# B&R Automation Studio project HISTest (part 2)

#### mbus_mast.var - Local variables
```iecst
(********************************************************************
 * COPYRIGHT -- Bernecker + Rainer
 ********************************************************************
 * Program: mbus_mast
 * File: mbus_mast.var
 * Author: Bernecker + Rainer
 * Created: February 17, 2010
 ********************************************************************
 * Local variables of program mbus_mast
 ********************************************************************)
VAR
	step : step_typ;
END_VAR
```

#### Action.st
```iecst
ACTION ActMbRtuMaster:

	CASE step OF

		MB_OPEN:

			MbMaster.MBMOpen_0.enable	:= TRUE;

			//MbMaster.MBMOpen_0.pDevice	:= ADR('IF1.ST2.IF1.ST3.IF1');  (* Device description string *)

			MbMaster.MBMOpen_0.pDevice	:= ADR('IF6.ST1.IF1');
			MbMaster.MBMOpen_0.pMode	:= ADR('/PHY=RS485 /PA=N /DB=8 /SB=1 /BD=19200');  (* Mode description string *)
			MbMaster.MBMOpen_0.pConfig	:= ADR('datamod');  (* Data object name *)
			MbMaster.MBMOpen_0.timeout	:= 2000;  (* Timeout in milliseconds (the value must be a multiple of 10 and >250ms) *)
			MbMaster.MBMOpen_0.ascii	:= 0;  (* 0 = RTU / 1 = ASCII *)

			MbMaster.MBMOpen_0();

			IF (MbMaster.MBMOpen_0.status = 0) AND (MbMaster.MBMOpen_0.ident <> 0) THEN
				step := MB_RUN;
				gSignalCheck.RS485_Check := TRUE;
			ELSIF MbMaster.MBMOpen_0.status = 65535 THEN
			ELSIF MbMaster.MBMOpen_0.status <> 0 THEN
				step := MB_ERROR;
			END_IF

		MB_RUN:

			(*When the command Auto is True the MBMbMaster FUB is executed, otherwise the MCMCmd FUB is executed*)
			IF (MbMaster.Auto = TRUE) THEN
				MbMaster.MBMaster_0.enable	:= TRUE;
				MbMaster.MBMaster_0.ident		:= MbMaster.MBMOpen_0.ident;
				MbMaster.MBMaster_0();

				IF (MbMaster.MBMaster_0.status = 65535) THEN
				ELSIF MbMaster.MBMaster_0.status <> 0 THEN
					step := MB_ERROR;
				END_IF

			ELSE
				MbMaster.MBMCmd_0.enable	:= TRUE;
				MbMaster.MBMCmd_0.ident		:= MbMaster.MBMOpen_0.ident;

				IF (MbMaster.ReadDataTrigger) THEN
					MbMaster.MBMCmd_0.mfc 		:= 3;
					MbMaster.MBMCmd_0.data		:= ADR(MbMaster.ReadData);
					MbMaster.MBMCmd_0.offset	:= 0;
				ELSIF(MbMaster.WriteDataTrigger)THEN
					MbMaster.MBMCmd_0.mfc 		:= 16;
					MbMaster.MBMCmd_0.data		:= ADR(MbMaster.WriteData);  (* address of data area *)
					MbMaster.MBMCmd_0.offset	:= 100;
				END_IF;
				MbMaster.MBMCmd_0.node		:= 1;  (* address of the slave station *)
				MbMaster.MBMCmd_0.len		:= 10;
				MbMaster.MBMCmd_0();
				IF (MbMaster.MBMCmd_0.status = 65535) THEN
				ELSIF (MbMaster.MBMCmd_0.status <> 0) THEN
					step := MB_ERROR;
				END_IF

			END_IF

		MB_CLOSE:

			MbMaster.MBMClose_0.enable	:= TRUE;
			MbMaster.MBMClose_0.ident	:= MbMaster.MBMOpen_0.ident;
			MbMaster.MBMClose_0();

			IF MbMaster.MBMClose_0.status = 0 THEN
				step := MB_OPEN;
			ELSIF MbMaster.MBMClose_0.status = 65535 THEN
			ELSIF MbMaster.MBMClose_0.status <> 0 THEN
				step := MB_ERROR;
			END_IF

		MB_ERROR:

			MbMaster.MBMaster_0.enable	:= FALSE;
			MbMaster.MBMaster_0();
			MbMaster.MBMCmd_0.enable	:= FALSE;
			MbMaster.MBMCmd_0();
			MbMaster.MBMClose_0.enable	:= FALSE;
			MbMaster.MBMClose_0();

			IF (MbMaster.MBMOpen_0.ident <> 0) THEN
				MbMaster.MBMOpen_0.enable	:= FALSE;
				MbMaster.MBMOpen_0();
				step := MB_CLOSE;
			ELSE
				step := MB_OPEN;
			END_IF

	END_CASE

END_ACTION
```

### Data object Logical/MbRTU/datamod (Simple)

#### datamod.dat
```
(********************************************************************
 * COPYRIGHT -- Bernecker + Rainer
 ********************************************************************
 * Data object: NewDataObject
 * File: datamod.dat
 * Author: Bernecker + Rainer
 * Created: February 15, 2010
 ********************************************************************
 * Data object file: datamod.dat
 ********************************************************************)

;--------------------
; Modbus command file
;--------------------
"MbMaster.WriteDataTrigger      ", 16, $01, "MbMaster.WriteData             ", 00100, 0010
"MbMaster.ReadDataTrigger       ", 03, $01, "MbMaster.ReadData              ", 00000, 0010
"MbMaster.ReadDataTrigger       ", 03, $01, "MbMaster.ReadData              ", 00001, 0002

;"LibDRVmbus.EventPV4            ", 16, $01, "LibDRVmbus.LocalPV4            ", 0000, 0003
;"LibDRVmbus.EventPV3            ", 03, $01, "LibDRVmbus.LocalPV3            ", 0000, 0003
; \_____________________________/	|    |    \_____________________________/    |      |
;			 	 |					|    |				  	 |				     |      |
;		   31 Characters		    |    |			   31 Characters  		     |      |_Number of coils or registers
;			 						|    |				   						 |_Offset of the Modbus Variables
;									|    |
;									|    |_Target Address of the slave station
;			 						|
;			 						|_ Modbus function
```

### Program Logical/DIOHandle (IEC)

#### Variables.var
```iecst
VAR
	ProRLY : BOOL;
	PRLY : BOOL;
	NRLY : BOOL;
	ProRLYAUX : BOOL;
	PRLYAUX : BOOL;
	NRLYAUX : BOOL;
	EMSRLYAUX : BOOL;
END_VAR
```

#### Main.st
```iecst
PROGRAM _INIT
	(* Insert code here *)
	Sys.ProRly	:= 0;
	Sys.PRly	:= 0;
	Sys.NRly	:= 0;
	ProRLYAUX 	:= 0;
	PRLYAUX 	:= 0;
	NRLYAUX 	:= 0;
	EMSRLYAUX	:= 0;
END_PROGRAM

PROGRAM _CYCLIC
	(* Insert code here *)
	IF Sys.ProRly = 1	 	THEN
		ProRLY := 1;
	ELSE
	   	ProRLY := 0;
	END_IF;

	IF Sys.PRly = 1	 	THEN
		PRLY := 1;
	ELSE
		PRLY := 0;
	END_IF;

	IF Sys.NRly = 1	 	THEN
		NRLY := 1;
	ELSE
		NRLY := 0;
	END_IF;

	(* DI Check *)
	IF ProRLYAUX = 1 THEN
		Sys.ProRlyAux :=1;
	ELSE
		Sys.ProRlyAux :=0;
	END_IF;

	IF PRLYAUX = 1 THEN
		Sys.PRlyAux :=1;
	ELSE
		Sys.PRlyAux :=0;
	END_IF;

	IF NRLYAUX = 1 THEN
		Sys.NRlyAux :=1;
	ELSE
		Sys.NRlyAux :=0;
	END_IF;

	IF EMSRLYAUX = 1 THEN
		Sys.EMSRlyAux :=0;
	ELSE
		Sys.EMSRlyAux :=1;
	END_IF;

END_PROGRAM

PROGRAM _EXIT
	(* Insert code here *)

END_PROGRAM
```

### Program Logical/PRAHandle (IEC)

#### Variables.var
```iecst
VAR
	WakeUpSig : BOOL;
	PRATimerProRlyOff : TON;
	PRATimerProRlyOn : TON;
	PRATimerWakeUpOff : TON;
	PRATimerSeqErr : TON;
	LoopCount : USINT;
	RackIndex : USINT;
	WakeCount : USINT;
	RackCount : USINT;
END_VAR
```

#### Action.st
```iecst
ACTION ATSystemReady:

	PRARackEnableCount := 0;

	FOR i := 0 TO 3 DO
		IF SubBMS_Calculator.BSA[i].Rack_State.Field.BSA_Divice_Status <> 0 THEN
			PRARackEnableCount := PRARackEnableCount + 1 ;
		END_IF;
	END_FOR;

	IF PRARackEnableCount = HMI.DeviceLoading.SetRackNum THEN
		PRARackReadyDone := TRUE;
	ELSE
		PRARackReadyDone := FALSE;
	END_IF;
END_ACTION

ACTION ATReset:
	IF Sys.ResetSig THEN

		SubBMS_Calculator.BMA[0].Field.BSA_Reset := TRUE;
		SubBMS_Calculator.BMA[1].Field.BSA_Reset := TRUE;
		SubBMS_Calculator.BMA[2].Field.BSA_Reset := TRUE;
		SubBMS_Calculator.BMA[3].Field.BSA_Reset := TRUE;

		PRARackResetCount := 0;

		FOR i := 0 TO 3 DO
			IF SubBMS_Calculator.BSA[i].Rack_AlarmState.Value[1] = 0 AND SubBMS_Calculator.BSA[i].Rack_State.Field.BSA_Divice_Status <> 0 THEN
				PRARackResetCount := PRARackResetCount + 1 ;
			END_IF;
		END_FOR;

		IF PRARackResetCount = HMI.DeviceLoading.SetRackNum THEN
			PRARackResetDone := TRUE;
			PRATimerReset.IN := FALSE;

			SubBMS_Calculator.BMA[0].Field.BSA_Reset := FALSE;
			SubBMS_Calculator.BMA[1].Field.BSA_Reset := FALSE;
			SubBMS_Calculator.BMA[2].Field.BSA_Reset := FALSE;
			SubBMS_Calculator.BMA[3].Field.BSA_Reset := FALSE;

		ELSE
			PRARackResetDone := FALSE;
		END_IF;

	END_IF;

END_ACTION

ACTION ATWakeUpSeq:

	CASE WakeUpStep OF
		vkWAKEUP_INITIAL:

			Sys.WakeUpSig := TRUE;
			PRATimerSeqErr.IN := TRUE;

			IF 	Sys.WakeUpSig THEN
				WakeUpStep := vkWAKEUP_RACK1;
			END_IF;

		vkWAKEUP_RACK1: // RACK1 WakeUp

			SubBMS_Calculator.BMA[0].Field.BSA_WakeUP := TRUE;

			IF SubBMS_Calculator.BSA[0].Rack_State.Field.BSA_Divice_Status = 4 THEN
				WakeUpStep := vkWAKEUP_RACK2;
			ELSIF	SubBMS_Calculator.BSA[0].Rack_State.Field.BSA_Divice_Status = 0 THEN
				WakeUpStep := vkWAKEUP_RACK2;
				SubBMS_Calculator.BMA[0].Field.BSA_WakeUP := FALSE;
			END_IF;

		vkWAKEUP_RACK2: // RACK2 WakeUp

			SubBMS_Calculator.BMA[1].Field.BSA_WakeUP := TRUE;

			IF SubBMS_Calculator.BSA[1].Rack_State.Field.BSA_Divice_Status = 4 THEN
				WakeUpStep := vkWAKEUP_RACK3;
			ELSIF	SubBMS_Calculator.BSA[1].Rack_State.Field.BSA_Divice_Status = 0 THEN
				WakeUpStep := vkWAKEUP_RACK3;
				SubBMS_Calculator.BMA[1].Field.BSA_WakeUP := FALSE;
			END_IF;

		vkWAKEUP_RACK3: // RACK3 WakeUp

				SubBMS_Calculator.BMA[2].Field.BSA_WakeUP := TRUE;

			IF SubBMS_Calculator.BSA[2].Rack_State.Field.BSA_Divice_Status = 4  THEN
				WakeUpStep := vkWAKEUP_RACK4;
			ELSIF	SubBMS_Calculator.BSA[2].Rack_State.Field.BSA_Divice_Status = 0 THEN
				WakeUpStep := vkWAKEUP_RACK4;
				SubBMS_Calculator.BMA[2].Field.BSA_WakeUP := FALSE;
			END_IF;

		vkWAKEUP_RACK4: // RACK4 WakeUp

				SubBMS_Calculator.BMA[3].Field.BSA_WakeUP := TRUE;

			IF SubBMS_Calculator.BSA[3].Rack_State.Field.BSA_Divice_Status = 4 THEN
				WakeUpStep := vkWAKEUP_NRLY;
			ELSIF	SubBMS_Calculator.BSA[3].Rack_State.Field.BSA_Divice_Status = 0 THEN
				WakeUpStep := vkWAKEUP_NRLY;
				SubBMS_Calculator.BMA[3].Field.BSA_WakeUP := FALSE;
			END_IF;

		vkWAKEUP_NRLY: // SYSTEM NEG RLY ON

			Sys.NRly := 1;

			PMS.BAR_DIO.Field.BRA_Nrelay_DO_Status := TRUE;

			IF Sys.NRlyAux = 1 THEN
				WakeUpStep := vkWAKEUP_PRORLY_ON;
			END_IF;

		vkWAKEUP_PRORLY_ON: // SYSTEM PRO RLY ON

			Sys.ProRly :=1;

			PMS.BAR_DIO.Field.BRA_ProRelay_DO_Status := TRUE;

			IF Sys.ProRlyAux = 1 THEN
				WakeUpStep := vkWAKEUP_DELAYTIME1;
			END_IF;

		vkWAKEUP_DELAYTIME1: // DELAY TIME
			// Timmer1 on
			PRATimerProRlyOn.IN := TRUE;

			IF PRATimerProRlyOn.Q = 1 THEN
				WakeUpStep := vkWAKEUP_PRLY;
			END_IF;

		vkWAKEUP_PRLY: // SYSTEM POS RLY ON

			Sys.PRly :=1;

			PMS.BAR_DIO.Field.BRA_Prelay_DO_Status := TRUE;

			IF Sys.PRlyAux = 1 THEN
				WakeUpStep := vkWAKEUP_DELAYTIME2;
			END_IF;

		vkWAKEUP_DELAYTIME2 : // DELAY TIME
			// Timer2 on
			PRATimerProRlyOff.IN := TRUE;
			IF PRATimerProRlyOff.Q = 1 THEN
				WakeUpStep := vkWAKEUP_PRORLY_OFF;
			END_IF;

		vkWAKEUP_PRORLY_OFF: // SYSTEM PRO RLY OFF

			Sys.ProRly := 0;

			PMS.BAR_DIO.Field.BRA_ProRelay_DO_Status := FALSE;

			IF Sys.ProRlyAux = 0 THEN
				WakeUpStep := vkWAKEUP_TIMERESET;
			END_IF;

		vkWAKEUP_TIMERESET : // Timer reset

			PRATimerProRlyOn.IN 	:= FALSE;
			PRATimerProRlyOff.IN 	:= FALSE;
			PRATimerSeqErr.IN 		:= FALSE;

			Sys.WakeUpSig 	:= FALSE;
			PRAWakeUpDone 	:= TRUE;

	END_CASE;

END_ACTION
ACTION ATStopSeq:

	PRAStopDone 	:= FALSE;

	CASE StopStep OF
		vkSTOP_INITIAL:

			Sys.StopSig := TRUE;
			PRATimerSeqErr.IN := TRUE;

			IF Sys.StopSig THEN
				StopStep := vkSTOP_NRLY;
			END_IF;

		vkSTOP_NRLY: // SYSTEM NEG RLY ON

			Sys.NRly := 0;

			PMS.BAR_DIO.Field.BRA_Nrelay_DO_Status := FALSE;

			IF Sys.NRlyAux = 0 THEN
				StopStep := vkSTOP_DELAYTIME1;
			END_IF;

		vkSTOP_DELAYTIME1: // DELAY TIME
			// Timmer1 on
			PRATimerProRlyOn.IN := TRUE;
			IF PRATimerProRlyOn.Q = 1 THEN
				StopStep := vkSTOP_PRLY;
			END_IF;

		vkSTOP_PRLY: // SYSTEM POS RLY ON

			Sys.PRly := 0;

			PMS.BAR_DIO.Field.BRA_Prelay_DO_Status := FALSE;

			IF Sys.PRlyAux = 0 THEN
				StopStep := vkSTOP_DELAYTIME2;
			END_IF;

		vkSTOP_DELAYTIME2 : // DELAY TIME
			// Timer2 on
			PRATimerProRlyOff.IN := TRUE;
			IF PRATimerProRlyOff.Q = 1 THEN
				StopStep := vkSTOP_RACK1;
			END_IF;

		vkSTOP_RACK1: // RACK1 WakeUp

			IF SubBMS_Calculator.BSA[0].Rack_State.Field.BSA_Divice_Status = 4 THEN
				SubBMS_Calculator.BMA[0].Field.BSA_WakeUP := FALSE;
			END_IF;

			IF SubBMS_Calculator.BSA[0].Rack_State.Field.BSA_Divice_Status = 3 OR SubBMS_Calculator.BSA[0].Rack_State.Field.BSA_Divice_Status = 0 THEN
				StopStep := vkSTOP_RACK2;
			END_IF;

		vkSTOP_RACK2: // RACK2 WakeUp

			IF SubBMS_Calculator.BSA[1].Rack_State.Field.BSA_Divice_Status = 4 THEN
				SubBMS_Calculator.BMA[1].Field.BSA_WakeUP := FALSE;
			END_IF;

			IF SubBMS_Calculator.BSA[1].Rack_State.Field.BSA_Divice_Status = 3 OR SubBMS_Calculator.BSA[1].Rack_State.Field.BSA_Divice_Status = 0 THEN
				StopStep := vkSTOP_RACK3;
			END_IF;

		vkSTOP_RACK3: // RACK3 WakeUp

			IF SubBMS_Calculator.BSA[2].Rack_State.Field.BSA_Divice_Status = 4 THEN
				SubBMS_Calculator.BMA[2].Field.BSA_WakeUP := FALSE;
			END_IF;

			IF SubBMS_Calculator.BSA[2].Rack_State.Field.BSA_Divice_Status = 3 OR SubBMS_Calculator.BSA[2].Rack_State.Field.BSA_Divice_Status = 0 THEN
				StopStep := vkSTOP_RACK4;
			END_IF;

		vkSTOP_RACK4: // RACK4 WakeUp

			IF SubBMS_Calculator.BSA[3].Rack_State.Field.BSA_Divice_Status = 4 THEN
				SubBMS_Calculator.BMA[3].Field.BSA_WakeUP := FALSE;
			END_IF;

			IF SubBMS_Calculator.BSA[3].Rack_State.Field.BSA_Divice_Status = 3 OR SubBMS_Calculator.BSA[3].Rack_State.Field.BSA_Divice_Status = 0 THEN
				StopStep := vkSTOP_TIMERESET;
			END_IF;

		vkSTOP_TIMERESET : // Timer reset

			PRATimerWakeUpOff.IN	:= FALSE;
			PRATimerSeqErr.IN		:= FALSE;

			PRAStopDone 	:= TRUE;

	END_CASE;

END_ACTION
```

#### Main.st
```iecst
PROGRAM _INIT
	(* Insert code here *)
	StateMa := 0;

	RackIndex := 0;
	RackEnable_Count := 0;

	PRATimerProRlyOn.IN		:= FALSE;
	PRATimerProRlyOn.PT 	:= T#500ms;
	PRATimerProRlyOff.IN	:= FALSE;
	PRATimerProRlyOff.PT	:= T#200ms;
	PRATimerWakeUpOff.IN 	:= FALSE;
	PRATimerWakeUpOff.PT 	:= T#100ms;
	PRATimerSeqErr.IN 		:= FALSE;
	PRATimerSeqErr.PT 		:= T#15s;

END_PROGRAM

PROGRAM _CYCLIC
	(* Insert code here *)

//		 EMS EDGE POSITIVE TRIGGER 		//

//	IF EDGEPOS(Sys.EMSRlyAux) THEN
//	  StateMa := 14;
//	END_IF;
//
//

	CASE StateMa OF
		vkSYSTEM_INITIAL: // INITIAL

			IF HMI.DeviceLoading.SetRackNum <> 0 THEN
	  			StateMa		:= vkSYSTEM_PROTECT_CHECK;
			END_IF;

		vkSYSTEM_PROTECT_CHECK:

			IF HMI.DialogBox.Protect_Trigger THEN
				StateMa		:= vkSUBBMS_TEMPCHECK;
			ELSE
				StateMa		:= vkSUBBMS_ALLRESET;
			END_IF;

			RackIndex := 0;
			RackEnable_Count := 0;

		vkSUBBMS_ALLRESET: // SUB BMS ALL RESET COMMAND ON

			FOR LoopCount := 0  TO RACK_MAXNUM_MINUS_1 DO
				SubBMS_Calculator.BMA[LoopCount].Field.BSA_Reset := TRUE;
			END_FOR;

			StateMa := vkSUBBMS_STATECHECK;

		vkSUBBMS_STATECHECK: // SUB BMS STATE CHECK AND SUB BMS RESET COMMAND OFF

			IF (SubBMS_Calculator.BMA[RackIndex].Field.BSA_Reset) THEN

				IF SubBMS_Calculator.BSA[RackIndex].Rack_State.Field.BSA_Divice_Status <> 0 THEN
					SubBMS_Calculator.BMA[RackIndex].Field.BSA_Reset := FALSE;

					RackEnable_Count	:= RackEnable_Count + 1;

				ELSIF SubBMS_Calculator.BSA[RackIndex].Rack_State.Field.BSA_Divice_Status = 0 THEN

					SubBMS_Calculator.BMA[RackIndex].Field.BSA_Reset := FALSE;

				END_IF;

			END_IF;

			RackIndex := RackIndex + 1;

			IF RackIndex >= 4 THEN

				RackIndex	:= 0;

				IF RackEnable_Count = (HMI.DeviceLoading.SetRackNum) THEN
					StateMa := vkSUBBMS_WAITCOMMAND;
				END_IF;

			END_IF;

		vkSUBBMS_TEMPCHECK:

			IF SubBMS_Calculator.BSA[RackIndex].Rack_State.Field.BSA_Divice_Status <> 0 THEN

				RackEnable_Count	:= RackEnable_Count + 1;

			ELSIF SubBMS_Calculator.BSA[RackIndex].Rack_State.Field.BSA_Divice_Status = 0 THEN

			END_IF;

			RackIndex := RackIndex + 1;

			IF RackIndex >= 4 THEN

				RackIndex	:= 0;

				IF RackEnable_Count = (HMI.DeviceLoading.SetRackNum) THEN
					StateMa := vkSUBBMS_WAITCOMMAND;
				END_IF;

			END_IF;

		vkSUBBMS_WAITCOMMAND: // WAIT COMMAND
			IF (PMS.PMS.Field.PMS_WakeUp_CMD) AND NOT(PMS.PMS.Field.PMS_FaultReset) AND NOT(PMS.PMS.Field.PMS_Po_RelayStatus) AND NOT(PMS.PMS.Field.PMS_Pro_RelayStatus) AND NOT(PMS.PMS.Field.PMS_Ne_RelayStatus) AND ABS(PMS.SysBatCal.Field.BSA_Curr_Total) <= 50 THEN
				StateMa := vkSUBBMS_FIRSTWAKEUP;
			END_IF;

		vkSUBBMS_FIRSTWAKEUP: // INITIATE FIRST WAKE-UP
			PRATimerSeqErr.IN := TRUE;

			RackIndex := 0;
			WakeCount := 0;

			FOR LoopCount := 0  TO RACK_MAXNUM_MINUS_1 DO
				IF HMI.RackEnable[LoopCount] THEN
					SubBMS_Calculator.BMA[LoopCount].Field.BSA_WakeUP 	:= TRUE;
					RackIndex											:=	LoopCount;
					EXIT;
				END_IF;

			END_FOR;
			//SubBMS_Calculator.BMA[RackIndex].Field.BSA_WakeUP := TRUE;

			StateMa := vkSUBBMS_WAKEUPSEQ;

		vkSUBBMS_WAKEUPSEQ: // CHECK CURRENT RACK STATUS

			IF SubBMS_Calculator.BSA[RackIndex].Rack_State.Field.BSA_Divice_Status = 4 THEN

				WakeCount := WakeCount + 1;

				IF RackIndex <= RACK_MAXNUM_MINUS_1-1 THEN
					FOR LoopCount := RackIndex + 1  TO RACK_MAXNUM_MINUS_1 DO
						IF HMI.RackEnable[LoopCount] THEN
							SubBMS_Calculator.BMA[LoopCount].Field.BSA_WakeUP 	:= TRUE;
							RackIndex											:=	LoopCount;
							EXIT;
						END_IF;

					END_FOR;
				END_IF;

				IF WakeCount = RackEnable_Count THEN
					StateMa := vkSYSTEM_NEGRLY_ON;
				ELSE
					IF WakeCount > RACK_MAXNUM_MINUS_1 THEN
						WakeCount	:= 0;
					END_IF;
				END_IF;
			END_IF;

		vkSYSTEM_NEGRLY_ON: // SYSTEM NEG RLY ON
			Sys.NRly := 1;

			PMS.BAR_DIO.Field.BRA_Nrelay_DO_Status := TRUE;

			IF Sys.NRlyAux = 1 THEN
	  			StateMa := vkSYSTEM_PRORLY_ON;
			END_IF;

		vkSYSTEM_PRORLY_ON: // SYSTEM PRO RLY ON
			Sys.ProRly :=1;

			PMS.BAR_DIO.Field.BRA_ProRelay_DO_Status := TRUE;

			IF Sys.ProRlyAux = 1 THEN
	  			StateMa := vkSYSTEM_RLYDELAY1;
			END_IF;

		vkSYSTEM_RLYDELAY1: // DELAY TIME
			// Timmer1 on
			PRATimerProRlyOn.IN := TRUE;
			IF PRATimerProRlyOn.Q = 1 THEN
				StateMa := vkSYSTEM_POSRLY_ON;
			END_IF;

		vkSYSTEM_POSRLY_ON: // SYSTEM POS RLY ON
			Sys.PRly :=1;

			PMS.BAR_DIO.Field.BRA_Prelay_DO_Status := TRUE;

			IF Sys.PRlyAux = 1 THEN
	  			StateMa := vkSYSTEM_RLYDELAY2;
			END_IF;

		vkSYSTEM_RLYDELAY2 : // DELAY TIME
			// Timer2 on
			PRATimerProRlyOff.IN := TRUE;
			IF PRATimerProRlyOff.Q = 1 THEN
				StateMa := vkSYSTEM_PRORLY_OFF;
			END_IF;

		vkSYSTEM_PRORLY_OFF: // SYSTEM PRO RLY OFF
			Sys.ProRly := 0;

			PMS.BAR_DIO.Field.BRA_ProRelay_DO_Status := FALSE;

			IF Sys.ProRlyAux = 0 THEN
	  			StateMa := vkSYSTEM_DELAY_RESET1;
			END_IF;

		vkSYSTEM_DELAY_RESET1 : // Timer reset

			PRATimerProRlyOn.IN 	:= FALSE;
			PRATimerProRlyOff.IN 	:= FALSE;
			PRATimerSeqErr.IN 		:= FALSE;

			StateMa := vkSYSTEM_RUN;

		vkSYSTEM_RUN: //RUN STATE (IDLE)

			IF NOT(PMS.PMS.Field.PMS_WakeUp_CMD) AND NOT(PMS.PMS.Field.PMS_FaultReset) AND NOT(PMS.PMS.Field.PMS_Po_RelayStatus) AND NOT(PMS.PMS.Field.PMS_Pro_RelayStatus) AND NOT(PMS.PMS.Field.PMS_Ne_RelayStatus) AND ABS(PMS.SysBatCal.Field.BSA_Curr_Total) <= 50 THEN
				StateMa := vkSYSTEM_NEGRLY_OFF;
			END_IF;
		vkSYSTEM_NEGRLY_OFF:

			PRATimerSeqErr.IN := TRUE;

			Sys.NRly := 0;

			PMS.BAR_DIO.Field.BRA_Nrelay_DO_Status := FALSE;

			IF Sys.NRlyAux = 0 THEN
				StateMa := vkSYSTEM_RLYDELAY3;
			END_IF;

		vkSYSTEM_RLYDELAY3 :
			PRATimerWakeUpOff.IN := TRUE;
			IF PRATimerWakeUpOff.Q = 1 THEN
				StateMa := vkSYSTEM_POSRLY_OFF;
			END_IF;

		vkSYSTEM_POSRLY_OFF :
			Sys.PRly := 0;

			PMS.BAR_DIO.Field.BRA_Prelay_DO_Status := FALSE;

			IF Sys.PRlyAux = 0 THEN
				StateMa := vkSUBBMS_FIRSTWAKEDOWN;
			END_IF;

		vkSUBBMS_FIRSTWAKEDOWN: // INITIATE FIRST WAKE-UP

			RackIndex := 0;
			WakeCount := 0;

			FOR LoopCount := 0  TO RACK_MAXNUM_MINUS_1 DO
				IF HMI.RackEnable[LoopCount] THEN
					SubBMS_Calculator.BMA[LoopCount].Field.BSA_WakeUP 	:= FALSE;
					RackIndex											:=	LoopCount;
					EXIT;
				END_IF;

			END_FOR;
			//SubBMS_Calculator.BMA[RackIndex].Field.BSA_WakeUP := TRUE;
			StateMa := vkSUBBMS_WAKEDOWNSEQ;

		vkSUBBMS_WAKEDOWNSEQ: // CHECK CURRENT RACK STATUS

			IF SubBMS_Calculator.BSA[RackIndex].Rack_State.Field.BSA_Divice_Status = 3 THEN

				WakeCount := WakeCount + 1;

				IF RackIndex <= RACK_MAXNUM_MINUS_1-1 THEN
					FOR LoopCount := RackIndex + 1  TO RACK_MAXNUM_MINUS_1 DO
						IF HMI.RackEnable[LoopCount] THEN
							SubBMS_Calculator.BMA[LoopCount].Field.BSA_WakeUP 	:= FALSE;
							RackIndex											:=	LoopCount;
							EXIT;
						END_IF;

					END_FOR;
				END_IF;

				IF WakeCount = RackEnable_Count THEN
					StateMa := vkSYSTEM_DELAY_RESET2;
				ELSE
					IF WakeCount > RACK_MAXNUM_MINUS_1 THEN
	 					WakeCount	:= 0;
					END_IF;

				END_IF;
			END_IF;
//			IF SubBMS_Calculator.BSA[RackIndex].Rack_State.Field.BSA_Divice_Status = 3 THEN
//				RackIndex := RackIndex + 1;
//
//				IF RackIndex <= Rack_Count THEN
//					SubBMS_Calculator.BMA[RackIndex].Field.BSA_WakeUP := FALSE;
//
//					StateMa := 18;
//				ELSE
//
//					StateMa := 19;
//				END_IF;
//			END_IF;

		vkSYSTEM_DELAY_RESET2 :
			PRATimerWakeUpOff.IN	:= FALSE;
			PRATimerSeqErr.IN		:= FALSE;

			StateMa := vkSUBBMS_WAITCOMMAND;

	END_CASE;

	// SYSTEM STATE SEQ AND RELAY CHECK

	CASE StateMa OF
		0..4: // RESET SEQ

			IF RackCount = HMI.DeviceLoading.SetRackNum THEN

				PMS.SysBatCal.Field.BSA_Divice_Status := 1; //INIT

			ELSE

				FOR LoopCount := 0  TO RACK_MAXNUM_MINUS_1 DO
					IF (HMI.RackEnable[LoopCount]) THEN
						IF SubBMS_Calculator.BSA[LoopCount].Rack_State.Field.BSA_Divice_Status = 3 OR  SubBMS_Calculator.BSA[LoopCount].Rack_State.Field.BSA_Divice_Status = 2 THEN
							RackCount := RackCount + 1 ;
						END_IF;
					END_IF;
				END_FOR;

				PMS.SysBatCal.Field.BSA_Divice_Status := 0; //READY

			END_IF;

			IF PMS.PMS.Field.PMS_Po_RelayStatus OR PMS.PMS.Field.PMS_Pro_RelayStatus OR PMS.PMS.Field.PMS_Ne_RelayStatus THEN
				PMS.BAR_Protect.Field.BRA_Prtct_RelayWelding := TRUE;
			ELSE
				PMS.BAR_Protect.Field.BRA_Prtct_RelayWelding := FALSE;
			END_IF;

		5:
			FOR LoopCount := 0 TO RACK_MAXNUM_MINUS_1 DO
				IF SubBMS_Calculator.BSA[LoopCount].Rack_State.Field.BSA_Neg_Rly OR SubBMS_Calculator.BSA[LoopCount].Rack_State.Field.BSA_Pos_Rly OR SubBMS_Calculator.BSA[LoopCount].Rack_State.Field.BSA_PreChar_Rly THEN
	  				PMS.BAR_Protect.Field.BRA_Prtct_RelayWelding := TRUE;
				END_IF;

			END_FOR;

			IF Sys.PRly OR Sys.NRly OR Sys.ProRly THEN
				PMS.BAR_Protect.Field.BRA_Prtct_RelayWelding := TRUE;
			ELSE
				PMS.BAR_Protect.Field.BRA_Prtct_RelayWelding := FALSE;
			END_IF;

		6..14: //WAKE UP SEQ
			PMS.SysBatCal.Field.BSA_Divice_Status := 2; //STANDBY

			IF PRATimerSeqErr.Q = 1 THEN
				//PMS.PMS_PAR_SEQErr := TRUE;
			END_IF;

		15:
			IF PMS.PMS.Field.PMS_Po_RelayStatus AND NOT(PMS.PMS.Field.PMS_Pro_RelayStatus) AND PMS.PMS.Field.PMS_Ne_RelayStatus THEN
				PMS.SysBatCal.Field.BSA_Divice_Status := 3; //RUN
			END_IF;

		16..21: //WAKE DOWN SEQ

			IF NOT(Sys.NRly) AND NOT(Sys.PRly) THEN
				PMS.SysBatCal.Field.BSA_Divice_Status := 2; //STANDBY
			END_IF;

			IF PRATimerSeqErr.Q = 1 THEN
				//PMS.PMS_PAR_SEQErr := TRUE;
			END_IF;

	END_CASE;

	PRATimerProRlyOn();
	PRATimerProRlyOff();
	PRATimerWakeUpOff();
	PRATimerSeqErr();

END_PROGRAM

PROGRAM _EXIT
	(* Insert code here *)

END_PROGRAM
```

### SubBMS.typ
```iecst
TYPE
	SubBMS_Calculator_type : 	STRUCT
		BMA : ARRAY[0..3]OF BMAN_typ;
		BSA : ARRAY[0..3]OF BSA_typ;
	END_STRUCT;
	SubBMS_type : 	STRUCT
		Rack1 : SubBMS_Rack_type;
		Rack2 : SubBMS_Rack_type;
		Rack3 : SubBMS_Rack_type;
		Rack4 : SubBMS_Rack_type;
	END_STRUCT;
	SubBMS_Rack_type : 	STRUCT
		BMA : BMAN_typ;
		BSA : BSA_typ;
	END_STRUCT;
	BMA_typ : 	STRUCT
		BMA1 : BMAN_typ;
		BMA2 : BMAN_typ;
		BMA3 : BMAN_typ;
		BMA4 : BMAN_typ;
	END_STRUCT;
	BMAN_typ : 	STRUCT
		Value : ARRAY[0..1]OF DWORD;
		Field : BMAN_Field_typ;
	END_STRUCT;
	BMAN_Field_typ : 	STRUCT
		BSA_WakeUP : BOOL;
		BSA_Mode : BOOL;
		BSA_Reset : BOOL;
		BSA_Cell_MinV : UINT;
		BSA_Cell_AGV : INT;
	END_STRUCT;
	BSA_typ : 	STRUCT
		BSA_Product : BSA_Product_typ;
		Rack_Calc : Rack_Calc_typ;
		Rack_State : Rack_State_typ;
		Rack_AlarmState : Rack_AlarmState_typ;
		Rack_PWRCalc : Rack_PWRCalc_typ;
		Rack_Cell_Vcalc : Rack_Cell_Vcalc_typ;
		Rack_Cell_Tcalc : Rack_Cell_Tcalc_typ;
		Rack_Cell_Pcalc : Rack_Cell_Pcalc_typ;
		Modul1_Info : ModulN_Info_typ;
		Modul2_Info : ModulN_Info_typ;
		Modul3_Info : ModulN_Info_typ;
		Modul4_Info : ModulN_Info_typ;
		Modul5_Info : ModulN_Info_typ;
		Modul6_Info : ModulN_Info_typ;
		Modul7_Info : ModulN_Info_typ;
	END_STRUCT;
	BSA_Product_typ : 	STRUCT
		Value : ARRAY[0..1]OF DWORD;
		Field : BSA_Product_Field_typ;
	END_STRUCT;
	Rack_Calc_typ : 	STRUCT
		Value : ARRAY[0..1]OF DWORD;
		Field : Rack_Calc_Field_typ;
	END_STRUCT;
	Rack_State_typ : 	STRUCT
		Value : ARRAY[0..1]OF DWORD;
		Field : Rack_State_Field_typ;
	END_STRUCT;
	Rack_AlarmState_typ : 	STRUCT
		Value : ARRAY[0..1]OF DWORD;
		Field : Rack_AlarmState_Fieild_typ;
	END_STRUCT;
	Rack_PWRCalc_typ : 	STRUCT
		Value : ARRAY[0..1]OF DWORD;
		Field : Rack_PWRCalc_Field_typ;
	END_STRUCT;
	Rack_Cell_Vcalc_typ : 	STRUCT
		Value : ARRAY[0..1]OF DWORD;
		Field : Rack_Cell_Vcalc_Field_typ;
	END_STRUCT;
	Rack_Cell_Tcalc_typ : 	STRUCT
		Value : ARRAY[0..1]OF DWORD;
		Field : Rack_Cell_Tcalc_Field_typ;
	END_STRUCT;
	Rack_Cell_Pcalc_typ : 	STRUCT
		Value : ARRAY[0..1]OF DWORD;
		Field : Rack_Cell_Pcalc_Field_typ;
	END_STRUCT;
	ModulN_Info_typ : 	STRUCT
		Value : ARRAY[0..1]OF DWORD;
		Field : ModulN_Info_Field_typ;
	END_STRUCT;
	BSA_Product_Field_typ : 	STRUCT
		BSA_Type : USINT;
		BSA_SW_Ver : USINT;
		BRA_Normal_Volt : REAL;
		BRA_Capacity : REAL;
		BSA_Serial : USINT;
		BSA_Parallel : USINT;
	END_STRUCT;
	Rack_Calc_Field_typ : 	STRUCT
		BRA_Volt_Total : REAL;
		BRA_Curr_Total : REAL;
		BRA_SOC : REAL;
		BRA_SOH : REAL;
	END_STRUCT;
	Rack_State_Field_typ : 	STRUCT
		BSA_Divice_Status : USINT;
		BSA_Protect_Status : USINT;
		BSA_Balance : BOOL;
		BSA_Neg_Rly : BOOL;
		BSA_Pos_Rly : BOOL;
		BSA_PreChar_Rly : BOOL;
		BSA_MSD_AUX : BOOL;
		BSA_EMG_SW : BOOL;
		BSA_Water_leak : BOOL;
		Not_Used1 : BOOL;
		Not_Used2 : USINT;
		BSA_Ah : INT;
		Not_Used3 : UINT;
	END_STRUCT;
	Rack_AlarmState_Fieild_typ : 	STRUCT
		warning : Rack_warningState_Field_typ;
		fault : Rack_FaultState_Field_typ;
		protect : Rack_ProtectState_Field_typ;
	END_STRUCT;
	Rack_warningState_Field_typ : 	STRUCT
		BSA_Wn_Dischager_OC : BOOL;
		BSA_Wn_Chager_OC : BOOL;
		BSA_Wn_SOC_OV : BOOL;
		BSA_Wn_SOC_Un : BOOL;
		BSA_Wn_OV : BOOL;
		BSA_Wn_UV : BOOL;
		BSA_Wn_Cell_OV : BOOL;
		BSA_Wn_Cell_UV : BOOL;
		BSA_Wn_Cell_UnbalV : BOOL;
		BSA_Wn_DisCharger_Cell_OT : BOOL;
		BSA_Wn_Charger_Cell_OT : BOOL;
		BSA_Wn_DisCharger_Cell_UT : BOOL;
		BSA_Wn_Charger_Cell_UT : BOOL;
		BSA_Wn_Cell_UnbalT : BOOL;
		BSA_Wn_Discharger_UnbaPWR : BOOL;
		BSA_Wn_Charger_UnbaPWR : BOOL;
	END_STRUCT;
	Rack_FaultState_Field_typ : 	STRUCT
		BSA_FLT_Dischager_OC : BOOL;
		BSA_FLT_Chager_OC : BOOL;
		BSA_FLT_SOC_OV : BOOL;
		BSA_FLT_SOC_Un : BOOL;
		BSA_FLT_OV : BOOL;
		BSA_FLT_UV : BOOL;
		BSA_FLT_Cell_OV : BOOL;
		BSA_FLT_Cell_UV : BOOL;
		BSA_FLT_Cell_UnbalV : BOOL;
		BSA_FLT_DisCharger_Cell_OT : BOOL;
		BSA_FLT_Charger_Cell_OT : BOOL;
		BSA_FLT_DisCharger_Cell_UT : BOOL;
		BSA_FLT_Charger_Cell_UT : BOOL;
		BSA_FLT_Cell_UnbalT : BOOL;
		BSA_FLT_Discharger_UnbaPWR : BOOL;
		BSA_FLT_Charger_UnbaPWR : BOOL;
	END_STRUCT;
	Rack_ProtectState_Field_typ : 	STRUCT
		BSA_Prtct_Dischager_OC : BOOL;
		BSA_Prtct_Chager_OC : BOOL;
		BSA_Prtct_SOC_OV : BOOL;
		BSA_Prtct_SOC_Un : BOOL;
		BSA_Prtct_OV : BOOL;
		BSA_Prtct_UV : BOOL;
		BSA_Prtct_Cell_OV : BOOL;
		BSA_Prtct_Cell_UV : BOOL;
		BSA_Prtct_Cell_UnbalV : BOOL;
		BSA_Prtct_DisCharger_Cell_OT : BOOL;
		BSA_Prtct_Charger_Cell_OT : BOOL;
		BSA_Prtct_DisCharger_Cell_UT : BOOL;
		BSA_Prtct_Charger_Cell_UT : BOOL;
		BSA_Prtct_Cell_UnbalT : BOOL;
		BSA_Prtct_Discharger_UnbaPWR : BOOL;
		BSA_Prtct_Charger_UnbaPWR : BOOL;
		BSA_Prtct_Rly_Err : BOOL;
		BSA_Prtct_IN_COM_Err : BOOL;
		BSA_Prtct_EX_COM_Err : BOOL;
		BSA_Prtct_CT_COM_Err : BOOL;
		BSA_Prtct_Water_Leak_Err : BOOL;
		BSA_Prtct_EMS_SW_Err : BOOL;
		Not_Used1 : BOOL;
		Not_Used2 : BOOL;
		Not_Used3 : USINT;
	END_STRUCT;
	Rack_PWRCalc_Field_typ : 	STRUCT
		BSA_CHAPWCont : REAL;
		BSA_DisCHAPWCont : REAL;
		BSA_CHAPWPeak : REAL;
		BSA_DisCHAPWPeak : REAL;
	END_STRUCT;
	Rack_Cell_Vcalc_Field_typ : 	STRUCT
		BSA_Cell_MaxV : REAL;
		BSA_Cell_MinV : REAL;
		BSA_Cell_AVGV : REAL;
		BSA_Cell_DeviV : UINT;
	END_STRUCT;
	Rack_Cell_Tcalc_Field_typ : 	STRUCT
		BSA_Cell_MaxT : REAL;
		BSA_Cell_MinT : REAL;
		BSA_Cell_AVGT : REAL;
		BSA_Cell_DeviT : REAL;
	END_STRUCT;
	Rack_Cell_Pcalc_Field_typ : 	STRUCT
		BSA_Cell_MaxV_Location : UINT;
		BSA_Cell_MinV_Location : UINT;
		BSA_Cell_MaxT_Location : UINT;
		BSA_Cell_MinT_Location : UINT;
	END_STRUCT;
	ModulN_Info_Field_typ : 	STRUCT
		Volt_Total : REAL;
		Agv_Volt : REAL;
		Agv_Temp : REAL;
		OPS_INITOK : BOOL;
		OPS_Fault : BOOL;
		OPS_Balan_On_OFF : BOOL;
		OPS_Waterleak_Err : BOOL;
		OPS_CellVolt_Err : BOOL;
		OPS_CellTemps_Err : BOOL;
		BATIC_Err : BOOL;
		CTCOM_Err : BOOL;
		OPS_MBCOM_Err : BOOL;
		Not_Used1 : BOOL;
		Not_Used2 : BOOL;
		Not_Used3 : BOOL;
		Not_Used4 : BOOL;
		Not_Used5 : BOOL;
		Not_Used6 : BOOL;
		Not_Used7 : BOOL;
	END_STRUCT;
END_TYPE
```

### HMI.typ
```iecst
TYPE
	HMI_typ : 	STRUCT
		Step : STEP_Enum;
		DeviceLoading : DeviceLoadingPanel_typ;
		RackEnable : ARRAY[0..RACK_MAXNUM_MINUS_1]OF BOOL;
		RackIndex : RackIndex_enum;
		Gauge : GaugePanel_typ;
		BatteryInfo : BATInfoPanel_typ;
		Module1Info : ModuleInfoPanel_typ;
		Module2Info : ModuleInfoPanel_typ;
		Module3Info : ModuleInfoPanel_typ;
		Module4Info : ModuleInfoPanel_typ;
		Module5Info : ModuleInfoPanel_typ;
		Module6Info : ModuleInfoPanel_typ;
		Module7Info : ModuleInfoPanel_typ;
		SystemRackInfo : SystemRackInfoPanel_typ;
		BSA_Divice_Status : STRING[20];
		DIOStatus : DIOStatusPanel_typ;
		ProtectStatus : ProtectStatusPanel_typ;
		SubBMS_AlarmTable : ARRAY[0..21]OF ALARM_Info_typ;
		AlarmTableIndex : AlarmTableIndex_enum;
		AdminLogin : AdminLogin_typ;
		AdminDeviceReset : BOOL;
		TrendData : TrendData_typ;
		DialogBox : DialogBox_typ;
	END_STRUCT;
	DeviceLoadingPanel_typ : 	STRUCT
		Trigger : BOOL;
		DeviceLoadingStep : USINT;
		RackLoading : USINT;
		DeviceLoading_Max : USINT;
		SetRackNum : USINT;
		LoadingText : STRING[40];
	END_STRUCT;
	GaugePanel_typ : 	STRUCT
		BRA_SOC : REAL;
		BRA_SOC_A : STRING[20];
		BRA_SOC_B : STRING[50];
		BRA_SOH : REAL;
		BRA_SOH_A : STRING[20];
		BRA_SOH_B : STRING[50];
		BRA_Volt_Total : REAL;
		BRA_Volt_Total_A : STRING[20];
		BRA_Volt_Total_B : STRING[50];
		BRA_Curr_Total : REAL;
		BRA_Curr_Total_A : STRING[20];
		BRA_Curr_Total_B : STRING[50];
	END_STRUCT;
	BATInfoPanel_typ : 	STRUCT
		BSA_Cell_MaxV : REAL;
		BSA_Cell_MinV : REAL;
		BSA_Cell_AVGV : REAL;
		BSA_Cell_DeviV : REAL;
		BSA_Cell_MaxT : REAL;
		BSA_Cell_MinT : REAL;
		BSA_Cell_AVGT : REAL;
		BSA_Cell_DeviT : REAL;
		BSA_Cell_MaxV_Rack_Location : STRING[20];
		BSA_Cell_MaxV_Cell_Location : STRING[20];
		BSA_Cell_MaxV_Location : STRING[20];
		BSA_Cell_MinV_Rack_Location : STRING[20];
		BSA_Cell_MinV_Cell_Location : STRING[20];
		BSA_Cell_MinV_Location : STRING[20];
		BSA_Cell_MaxT_Rack_Location : STRING[20];
		BSA_Cell_MaxT_Cell_Location : STRING[20];
		BSA_Cell_MaxT_Location : STRING[20];
		BSA_Cell_MinT_Rack_Location : STRING[20];
		BSA_Cell_MinT_Cell_Location : STRING[20];
		BSA_Cell_MinT_Location : STRING[20];
	END_STRUCT;
	ModuleInfoPanel_typ : 	STRUCT
		Volt_Total_A : STRING[20];
		Volt_Total_B : STRING[20];
		OPS_Fault : STRING[20];
		CTCOM_Err : STRING[20];
		OPS_MBCOM_Err : STRING[20];
	END_STRUCT;
	SystemRackInfoPanel_typ : 	STRUCT
		RACK_State : ARRAY[0..3]OF STRING[20];
		RACK_BRA_Volt_Total : ARRAY[0..3]OF STRING[20];
		RACK_BRA_Curr_Total : ARRAY[0..3]OF STRING[20];
		RACK_BRA_Total : ARRAY[0..3]OF STRING[20];
	END_STRUCT;
	DIOStatusPanel_typ : 	STRUCT
		BSA_EMS : STRING[20];
		BSA_OffGas : STRING[20];
		BSA_Water_leak : STRING[20];
		BSA_Neg_Rly : STRING[20];
		BSA_PreChar_Rly : STRING[20];
		BSA_Pos_Rly : STRING[20];
	END_STRUCT;
	ProtectStatusPanel_typ : 	STRUCT
		BSA_Charge_OC : STRING[20];
		BSA_Discharge_OC : STRING[20];
		BSA_OC : STRING[20];
		BSA_SOC_OV : STRING[20];
		BSA_SOC_Un : STRING[20];
		BSA_OV : STRING[20];
		BSA_UV : STRING[20];
		BSA_Cell_OV : STRING[20];
		BSA_Cell_UV : STRING[20];
		BSA_Cell_UnbalV : STRING[20];
		BSA_DisCharger_Cell_OT : STRING[20];
		BSA_Charger_Cell_OT : STRING[20];
		BSA_DisCharger_Cell_UT : STRING[20];
		BSA_Charger_Cell_UT : STRING[20];
		BSA_Cell_UnbalT : STRING[20];
		BSA_Discharge_Unbal_PWR : STRING[20];
		BSA_Charge_Unbal_PWR : STRING[20];
		BSA_Prtct_Peak_OP : STRING[20];
		BSA_Prtct_Continuously_OP : STRING[20];
		BSA_Prtct_IN_COM_Err : STRING[20];
		BSA_Prtct_EX_COM_Err : STRING[20];
		BSA_Prtct_Rly_Err : STRING[20];
		BSA_Prtct_Water_Leak_Err : STRING[20];
		BRA_Prtct_InsulationReg : STRING[20];
		BRA_Prtct_MDSFuse : STRING[20];
		BSA_Prtct_CoolingSystem : STRING[20];
	END_STRUCT;
	Alarm_typ : 	STRUCT
		Warning : ARRAY[0..21]OF ALARM_Info_typ;
		Fault : ARRAY[0..21]OF ALARM_Info_typ;
		Protect : ARRAY[0..21]OF ALARM_Info_typ;
	END_STRUCT;
	ALARM_Info_typ : 	STRUCT
		Name : STRING[30];
		InitialTime : STRING[15];
		RecentTime : STRING[15];
		ClearTime : STRING[15];
		Count : USINT;
	END_STRUCT;
	Dialog_typ : 	STRUCT
		Name : STRING[30];
		Trigger : BOOL;
	END_STRUCT;
	AdminLogin_typ : 	STRUCT
		Authority : LoginStatusEnum;
		Input_Button : STRING[1];
		Password_Internal : STRING[16];
		Password_External : STRING[16];
	END_STRUCT;
	TrendData_typ : 	STRUCT
		Voltage : REAL;
		Current : REAL;
	END_STRUCT;
	DialogBox_typ : 	STRUCT
		LoadingError_Trigger : BOOL;
		BuzzerOFF_Trigger : BOOL;
		Protect_Trigger : BOOL;
		ProtectName : STRING[30];
	END_STRUCT;
	STEP_Enum :
		(
		vkINITIAL := 0,
		vkBOOTING := 1,
		vkSYSTEM := 2,
		vkRACK1 := 3,
		vkRACK2 := 4,
		vkRACK3 := 5,
		vkRACK4 := 6,
		vkADMINISTRATOR := 13,
		vkALARMHISTORY := 14,
		vkLOADINGERROR := 15,
		vkPROTECTERROR := 16,
		vkUSERTEST := 20
		);
	RackIndex_enum :
		(
		vkRACKNUM1 := 0,
		vkRACKNUM2 := 1,
		vkRACKNUM3 := 2,
		vkRACKNUM4 := 3
		);
	AlarmTableIndex_enum :
		(
		vkWarning := 0,
		vkFault := 1,
		vkProtect := 2
		);
	LoginStatusEnum :
		(
		USER := 0,
		ADMIN := 1
		);
END_TYPE
```

### PMS_CAN.typ
```iecst
TYPE
	PMS_typ : 	STRUCT
		PMS : PMS_type;
		SysBatProduct : SysBatProduct_typ;
		SysBatCal : SysBatCal_typ;
		SysBatPWR : SysBatPWR_typ;
		SysCellVolt : SysCellVolt_typ;
		SysCellTemps : SysCellTemps_typ;
		SysCellV_TPos : SysCellV_TPos_typ;
		SysBatProtect : SysBatProtect_typ;
		SysBatDIO : SysBatDIO_typ;
		BRACal : BRACal_typ;
		BRAPWR_A : BRAPWR_A_typ;
		BRAPWR_B : BRAPWR_B_typ;
		BRACellV : BRACellV_typ;
		BRACellT : BRACellT_typ;
		BRACellDiv : BRACellDiv_typ;
		BRA_VTPos : BRA_VTPos_typ;
		BAR_Alarm : BAR_Alarm_typ;
		BAR_Protect : BAR_Protect_typ;
		BAR_DIO : BAR_DIO_typ;
	END_STRUCT;
	PMS_type : 	STRUCT
		Value : ARRAY[0..1]OF DWORD;
		Field : PMS_Field_typ;
	END_STRUCT;
	SysBatProduct_typ : 	STRUCT
		Value : ARRAY[0..1]OF DWORD;
		Field : SysBatProduct_Field_typ;
	END_STRUCT;
	SysBatCal_typ : 	STRUCT
		Value : ARRAY[0..1]OF DWORD;
		Field : SysBatCal_Field_typ;
	END_STRUCT;
	SysBatPWR_typ : 	STRUCT
		Value : ARRAY[0..1]OF DWORD;
		Field : SysBatPWR_Field_typ;
	END_STRUCT;
	SysCellVolt_typ : 	STRUCT
		Value : ARRAY[0..1]OF DWORD;
		Field : SysCellVolt_Field_typ;
	END_STRUCT;
	SysCellTemps_typ : 	STRUCT
		Value : ARRAY[0..1]OF DWORD;
		Field : SysCellTemps_Field_typ;
	END_STRUCT;
	SysCellV_TPos_typ : 	STRUCT
		Value : ARRAY[0..1]OF DWORD;
		Field : SysCellV_TPos_Field_typ;
	END_STRUCT;
	SysBatProtect_typ : 	STRUCT
		Value : ARRAY[0..1]OF DWORD;
		Field : SysBatProtect_Field_typ;
	END_STRUCT;
	SysBatDIO_typ : 	STRUCT
		Value : ARRAY[0..1]OF DWORD;
		Field : SysBatDIO_Field_typ;
	END_STRUCT;
	BRACal_typ : 	STRUCT
		Value : ARRAY[0..1]OF DWORD;
		Field : BRACal_Field_typ;
	END_STRUCT;
	BRAPWR_A_typ : 	STRUCT
		Value : ARRAY[0..1]OF DWORD;
		Field : BRAPWR_A_Field_typ;
	END_STRUCT;
	BRAPWR_B_typ : 	STRUCT
		Value : ARRAY[0..1]OF DWORD;
		Field : BRAPWR_B_Field_typ;
	END_STRUCT;
	BRACellV_typ : 	STRUCT
		Value : ARRAY[0..1]OF DWORD;
		Field : BRACellV_Field_typ;
	END_STRUCT;
	BRACellT_typ : 	STRUCT
		Value : ARRAY[0..1]OF DWORD;
		Field : BRACellT_Field_typ;
	END_STRUCT;
	BRACellDiv_typ : 	STRUCT
		Value : ARRAY[0..1]OF DWORD;
		Field : BRACellDiv_Field_typ;
	END_STRUCT;
	BRA_VTPos_typ : 	STRUCT
		Value : ARRAY[0..1]OF DWORD;
		Field : BRA_VTPos_Field_typ;
	END_STRUCT;
	BAR_Alarm_typ : 	STRUCT
		Value : ARRAY[0..1]OF DWORD;
		Field : BAR_Alarm_Field_typ;
	END_STRUCT;
	BAR_Protect_typ : 	STRUCT
		Value : ARRAY[0..1]OF DWORD;
		Field : BAR_Protect_Field_typ;
	END_STRUCT;
	BAR_DIO_typ : 	STRUCT
		Value : ARRAY[0..1]OF DWORD;
		Field : BAR_DIO_Field_typ;
	END_STRUCT;
	PMS_Field_typ : 	STRUCT
		PMS_WakeUp_CMD : BOOL;
		PMS_POWER_CMD : BOOL;
		PMS_FaultReset : BOOL;
		PMS_Po_RelayStatus : BOOL;
		PMS_Pro_RelayStatus : BOOL;
		PMS_Ne_RelayStatus : BOOL;
	END_STRUCT;
	SysBatProduct_Field_typ : 	STRUCT
		BSA_Production_Year : UINT;
		BSA_Production_Type : USINT;
		BSA_Production_Num : USINT;
		BSA_Production_VER : USINT;
		BSA_Production_BSA_Serial : USINT;
		BSA_Production_BSA_Parallel : USINT;
	END_STRUCT;
	SysBatCal_Field_typ : 	STRUCT
		BSA_Volt_Total : REAL;
		BSA_Curr_Total : REAL;
		BSA_SOC : REAL;
		BSA_Divice_Status : UINT;
	END_STRUCT;
	SysBatPWR_Field_typ : 	STRUCT
		BSA_Cont_Charge_Power_Limit : REAL;
		BSA_Peak_Charge_Power_Limit : REAL;
		BSA_Cont_Discharge_Power_Limit : REAL;
		BSA_Peak_Discharge_Power_Limit : REAL;
	END_STRUCT;
	SysCellVolt_Field_typ : 	STRUCT
		BSA_Cell_MaxV : REAL;
		BSA_Cell_MinV : REAL;
		BSA_Cell_AVGV : REAL;
		BSA_Cell_DeviV : REAL;
	END_STRUCT;
	SysCellTemps_Field_typ : 	STRUCT
		BSA_Cell_MaxT : REAL;
		BSA_Cell_MinT : REAL;
		BSA_Cell_AVGT : REAL;
		BSA_Cell_DeviT : REAL;
	END_STRUCT;
	SysCellV_TPos_Field_typ : 	STRUCT
		BSA_Rack_MaxV_Location : USINT;
		BSA_Cell_MaxV_Location : USINT;
		BSA_Rack_MinV_Location : USINT;
		BSA_Cell_MinV_Location : USINT;
		BSA_Rack_MaxT_Location : USINT;
		BSA_Cell_MaxT_Location : USINT;
		BSA_Rack_MinT_Location : USINT;
		BSA_Cell_MinT_Location : USINT;
	END_STRUCT;
	SysBatProtect_Field_typ : 	STRUCT
		BSA_Alarm_OC : BOOL;
		BSA_Alarm_SOC_OV : BOOL;
		BSA_Alarm_SOC_UN : BOOL;
		BSA_Alarm_OV : BOOL;
		BSA_Alarm_UV : BOOL;
		BSA_Alarm_Cell_OV : BOOL;
		BSA_Alarm_Cell_UV : BOOL;
		BSA_Alarm_Cell_UnBalaV : BOOL;
		BSA_Alarm_Discharger_Cell_OT : BOOL;
		BSA_Alarm_Charger_Cell_OT : BOOL;
		BSA_Alarm_Discharger_Cell_UT : BOOL;
		BSA_Alarm_Charger_Cell_UT : BOOL;
		BSA_Alarm_Cell_UnBalaT : BOOL;
		BSA_Alarm_Continuously_OP : BOOL;
		BSA_Alarm_Peak_OP : BOOL;
		BSA_Fault_OC : BOOL;
		BSA_Fault_SOC_OV : BOOL;
		BSA_Fault_SOC_UN : BOOL;
		BSA_Fault_OV : BOOL;
		BSA_Fault_UV : BOOL;
		BSA_Fault_Cell_OV : BOOL;
		BSA_Fault_Cell_UV : BOOL;
		BSA_Fault_Cell_UnBalaV : BOOL;
		BSA_Fault_Discharger_Cell_OT : BOOL;
		BSA_Fault_Charger_Cell_OT : BOOL;
		BSA_Fault_Discharger_Cell_UT : BOOL;
		BSA_Fault_Charger_Cell_UT : BOOL;
		BSA_Fault_Cell_UnBalaT : BOOL;
		BSA_Fault_Continuously_OP : BOOL;
		BSA_Fault_Peak_OP : BOOL;
		BSA_Prtct_OC : BOOL;
		BSA_Prtct_SOC_OV : BOOL;
		BSA_Prtct_SOC_UN : BOOL;
		BSA_Prtct_OV : BOOL;
		BSA_Prtct_UV : BOOL;
		BSA_Prtct_Cell_OV : BOOL;
		BSA_Prtct_Cell_UV : BOOL;
		BSA_Prtct_Cell_UnBalaV : BOOL;
		BSA_Prtct_Discharger_Cell_OT : BOOL;
		BSA_Prtct_Charger_Cell_OT : BOOL;
		BSA_Prtct_Discharger_Cell_UT : BOOL;
		BSA_Prtct_Charger_Cell_UT : BOOL;
		BSA_Prtct_Cell_UnBalaT : BOOL;
		BSA_Prtct_Continuously_OP : BOOL;
		BSA_Prtct_Peak_OP : BOOL;
		BSA_Prtct_InternalCOM : BOOL;
		BSA_Prtct_ExternalCOM : BOOL;
		BSA_Prtct_RelayWelding : BOOL;
		BSA_Prtct_WaterLeak : BOOL;
		BSA_Prtct_InsulationReg : BOOL;
		BSA_Prtct_MDSFuse : BOOL;
		BSA_Prtct_Cooling_System : BOOL;
	END_STRUCT;
	SysBatDIO_Field_typ : 	STRUCT
		BSA_Prelay_DO_Status : BOOL;
		BSA_Nrelay_DO_Status : BOOL;
		BSA_ProRelay_DO_Status : BOOL;
		BSA_Buzzer_DO_Status : BOOL;
		BSA_PowerLamp_DO_Status : BOOL;
		BSA_DO_Spare06 : BOOL;
		BSA_DO_Spare07 : BOOL;
		BSA_DO_Spare08 : BOOL;
		BSA_DO_Spare09 : BOOL;
		BSA_DO_Spare10 : BOOL;
		BSA_DO_Spare11 : BOOL;
		BSA_DO_Spare12 : BOOL;
		BSA_PRelayAUX_DI_Status : BOOL;
		BSA_NRelayAUX_DI_Status : BOOL;
		BSA_EMGSwitch_DI_Status : BOOL;
		BSA_CoolingSystem_DI_Status : BOOL;
		BSA_MDS_DI_Status : BOOL;
		BSA_DI_Spare06 : BOOL;
		BSA_DI_Spare07 : BOOL;
		BSA_DI_Spare08 : BOOL;
		BSA_DI_Spare09 : BOOL;
		BSA_DI_Spare10 : BOOL;
		BSA_DI_Spare11 : BOOL;
		BSA_DI_Spare12 : BOOL;
		BSA_SOH : REAL;
	END_STRUCT;
	BRACal_Field_typ : 	STRUCT
		BRA_Rack_Num : UINT;
		BRA_Volt_Total : REAL;
		BRA_Curr_Total : REAL;
		BRA_SOC : REAL;
	END_STRUCT;
	BRAPWR_A_Field_typ : 	STRUCT
		BRA_Rack_Num : UINT;
		BRA_SOH : REAL;
		BRA_CONT_CHA_PWR_Limit : REAL;
		BRA_Peak_CHA_PWR_Limit : REAL;
	END_STRUCT;
	BRAPWR_B_Field_typ : 	STRUCT
		BRA_Rack_Num : UINT;
		BRA_CONT_DisCHA_PWR_Limit : REAL;
		BRA_Peak_DisCHA_PWR_Limit : REAL;
	END_STRUCT;
	BRACellV_Field_typ : 	STRUCT
		BRA_Rack_Num : UINT;
		BRA_Cell_Max_Voltage : REAL;
		BRA_Cell_Min_Voltage : REAL;
		BRA_Cell_AGV_Voltage : REAL;
	END_STRUCT;
	BRACellT_Field_typ : 	STRUCT
		BRA_Rack_Num : UINT;
		BRA_Cell_Max_Temperature : REAL;
		BRA_Cell_Min_Temperature : REAL;
		BRA_Cell_AGV_Temperature : REAL;
	END_STRUCT;
	BRACellDiv_Field_typ : 	STRUCT
		BRA_Rack_Num : UINT;
		BRA_Cell_DIV_Voltage : REAL;
		BRA_Cell_DIV_Temperature : REAL;
	END_STRUCT;
	BRA_VTPos_Field_typ : 	STRUCT
		BRA_Rack_Num : UINT;
		BRA_Max_Cell_V_Location : USINT;
		BRA_Min_Cell_V_Location : USINT;
		BRA_Max_Cell_T_Location : USINT;
		BRA_Min_Cell_T_Location : USINT;
	END_STRUCT;
	BAR_Alarm_Field_typ : 	STRUCT
		BRA_Rack_Num : UINT;
		BRA_Alarm_OC : BOOL;
		BRA_Alarm_SOC_OV : BOOL;
		BRA_Alarm_SOC_UN : BOOL;
		BRA_Alarm_OV : BOOL;
		BRA_Alarm_UV : BOOL;
		BRA_Alarm_Cell_OV : BOOL;
		BRA_Alarm_Cell_UV : BOOL;
		BRA_Alarm_Cell_UnBalaV : BOOL;
		BRA_Alarm_Discharger_Cell_OT : BOOL;
		BRA_Alarm_Charger_Cell_OT : BOOL;
		BRA_Alarm_Discharger_Cell_UT : BOOL;
		BRA_Alarm_Charger_Cell_UT : BOOL;
		BRA_Alarm_Cell_UnBalaT : BOOL;
		BRA_Alarm_Continuously_OP : BOOL;
		BRA_Alarm_Peak_OP : BOOL;
		BRA_Fault_OC : BOOL;
		BRA_Fault_SOC_OV : BOOL;
		BRA_Fault_SOC_UN : BOOL;
		BRA_Fault_OV : BOOL;
		BRA_Fault_UV : BOOL;
		BRA_Fault_Cell_OV : BOOL;
		BRA_Fault_Cell_UV : BOOL;
		BRA_Fault_Cell_UnBalaV : BOOL;
		BRA_Fault_Discharger_Cell_OT : BOOL;
		BRA_Fault_Charger_Cell_OT : BOOL;
		BRA_Fault_Discharger_Cell_UT : BOOL;
		BRA_Fault_Charger_Cell_UT : BOOL;
		BRA_Fault_Cell_UnBalaT : BOOL;
		BRA_Fault_Continuously_OP : BOOL;
		BRA_Fault_Peak_OP : BOOL;
	END_STRUCT;
	BAR_Protect_Field_typ : 	STRUCT
		BRA_Rack_Num : UINT;
		BRA_Prtct_OC : BOOL;
		BRA_Prtct_SOC_OV : BOOL;
		BRA_Prtct_SOC_UN : BOOL;
		BRA_Prtct_OV : BOOL;
		BRA_Prtct_UV : BOOL;
		BRA_Prtct_Cell_OV : BOOL;
		BRA_Prtct_Cell_UV : BOOL;
		BRA_Prtct_Cell_UnBalaV : BOOL;
		BRA_Prtct_Discharger_Cell_OT : BOOL;
		BRA_Prtct_Charger_Cell_OT : BOOL;
		BRA_Prtct_Discharger_Cell_UT : BOOL;
		BRA_Prtct_Charger_Cell_UT : BOOL;
		BRA_Prtct_Cell_UnBalaT : BOOL;
		BRA_Prtct_Continuously_OP : BOOL;
		BRA_Prtct_Peak_OP : BOOL;
		BRA_Prtct_InternalCOM : BOOL;
		BRA_Prtct_ExternalCOM : BOOL;
		BRA_Prtct_RelayWelding : BOOL;
		BRA_Prtct_WaterLeak : BOOL;
		BRA_Prtct_InsulationReg : BOOL;
		BRA_Prtct_MDSFuse : BOOL;
		BRA_Prtct_CoolingSystem : BOOL;
	END_STRUCT;
	BAR_DIO_Field_typ : 	STRUCT
		BRA_Rack_Num : UINT;
		BRA_Prelay_DO_Status : BOOL;
		BRA_Nrelay_DO_Status : BOOL;
		BRA_ProRelay_DO_Status : BOOL;
		BRA_PowerLamp_DO_Status : BOOL;
		BRA_Buzzer_DO_Status : BOOL;
		BRA_PRelayAUX_DI_Status : BOOL;
		BRA_NRelayAUX_DI_Status : BOOL;
		BRA_EMGSwitch_DI_Status : BOOL;
		BRA_MDS_DI_Status : BOOL;
		BRA_Waterleak_Dete_MD1 : BOOL;
		BRA_Waterleak_Dete_MD2 : BOOL;
		BRA_Waterleak_Dete_MD3 : BOOL;
		BRA_Waterleak_Dete_MD4 : BOOL;
		BRA_Waterleak_Dete_MD5 : BOOL;
		BRA_Waterleak_Dete_MD6 : BOOL;
		BRA_Waterleak_Dete_MD7 : BOOL;
	END_STRUCT;
END_TYPE
```

### LAMP.typ
```iecst
TYPE
	LAMP_typ : 	STRUCT
		SW_B : BOOL;
	END_STRUCT;
END_TYPE
```

### Variables.var
```iecst
VAR CONSTANT
	PASSWORD : STRING[16] := '1234';
	RACK1 : USINT := 0;
	RACK2 : USINT := 1;
	RACK3 : USINT := 2;
	RACK4 : USINT := 3;
	RACK_MAXNUM : USINT := 4;
	RACK_MAXNUM_MINUS_1 : USINT := RACK_MAXNUM-1;
END_VAR
(*Insert your comment here.*)
(*Insert your comment here.*)
(*Insert your comment here.*)
VAR
	SubBMS : SubBMS_type;
	SubBMS_Sim : SubBMS_type;
	SubBMS_Calculator : SubBMS_Calculator_type;
	Rack_HMI : BSA_typ;
END_VAR
(*Insert your comment here.*)
(*Insert your comment here.*)
(*Insert your comment here.*)
VAR
	HMI : HMI_typ;
END_VAR
VAR RETAIN
	HMI_Alarm : Alarm_typ;
	HMI_AlarmName : ARRAY[0..21] OF STRING[30];
END_VAR
VAR
	HMI_Dialog : Dialog_typ;
END_VAR
(*Insert your comment here.*)
(*Insert your comment here.*)
(*Insert your comment here.*)
VAR
	PMS : PMS_typ;
	System_HMI : PMS_typ;
END_VAR
(*Insert your comment here.*)
(*Insert your comment here.*)
(*Insert your comment here.*)
VAR
	LAMP : LAMP_typ;
END_VAR
```

### Program Logical/Source/LAMPSeq/Lamp_SW_B (IEC)

#### Main.st
```iecst
PROGRAM _INIT
	(* Insert code here *)

END_PROGRAM

PROGRAM _CYCLIC
	(* Insert code here *)

	IF Sys.NRlyAux AND Sys.PRlyAux AND NOT(Sys.ProRlyAux) THEN
		LAMP.SW_B := TRUE;
	ELSE
		IF LAMP.SW_B THEN
			LAMP.SW_B := FALSE;
		ELSE
			LAMP.SW_B := TRUE;
		END_IF;
	END_IF;

END_PROGRAM

PROGRAM _EXIT
	(* Insert code here *)

END_PROGRAM
```

### Program Logical/Source/SubBMS_CAN/CANRxSubBMS (IEC)

#### ArCanReceive.st - Cyclic code
```iecst
PROGRAM _INIT

	ActArCanReceiver;
	ArCanReceiver.enable				:= TRUE;
	ArCanReceiver.receiverDeviceName 	:= 'IF7';       (* for X20CP0482 CPU *)
	ArCanReceiver.id					:= 16#600;
	//	ArCanReceiver.idMask				:= arCAN_RECEIVE_ALL;  // or configure IDMask
	ArCanReceiver.idMask				:= 16#600 ;  // or configure IDMask
	ArCanReceiver.format				:= arCAN_11BIT;  // or arCAN_29BIT
	ArCanReceiver.queueSize				:= 256;
	ArCanReceiver.ArCanSetBitTimingRegisters_0.Register0 := 0;
	ArCanReceiver.ArCanSetBitTimingRegisters_0.Register1 := 16#1C;

	(**********************	 CAN Baud rate Register Value	*************************)
	(********************************************************************************)
	(* 	  1 000 000 bit/s    >>		Register0 = 16#00	||		Register1 = 16#14	*)
	(* 		800 000 bit/s    >>		Register0 = 16#00	||		Register1 = 16#16	*)
	(* 		500 000 bit/s    >>		Register0 = 16#00	||		Register1 = 16#1C	*)
	(* 		250 000 bit/s    >>		Register0 = 16#01	||		Register1 = 16#1C	*)
	(* 		125 000 bit/s    >>		Register0 = 16#03	||		Register1 = 16#1C	*)
	(* 		100 000 bit/s    >>		Register0 = 16#04	||		Register1 = 16#1C	*)
	(* 		050 000 bit/s    >>		Register0 = 16#09	||		Register1 = 16#1C	*)
	(* 		020 000 bit/s    >>		Register0 = 16#18	||		Register1 = 16#1C	*)
	(* 		010 000 bit/s    >>		Register0 = 16#31	||		Register1 = 16#1C	*)
	(********************************************************************************)
	(********************************************************************************)

END_PROGRAM

PROGRAM _CYCLIC
	IF CmdSim THEN

		(*ActSimulation;*)
		memcpy(ADR(SubBMS), ADR(SubBMS_Sim), SIZEOF(SubBMS));

	ELSE
		ActArCanReceiver;
		(***********************************************************)
		(* Customize the received data *)
		// ArCanReceiver.ArCanReceiver_0.ReceivedFrame; //Data received
		IF (ArCanReceiver.ArCanReceiver_0.NewDataValid) THEN

			CASE ArCanReceiver.ArCanReceiver_0.ReceivedFrame.ID OF

				16#600..16#60E: // RACK 1

				//0 : BMS
				IF ArCanReceiver.ArCanReceiver_0.ReceivedFrame.ID = 16#600 THEN

					memcpy(ADR(SubBMS.Rack1.BSA.BSA_Product.Value), ADR(ArCanReceiver.ArCanReceiver_0.ReceivedFrame.Data), SIZEOF(SubBMS.Rack1.BSA.BSA_Product.Value));

				END_IF;
				IF ArCanReceiver.ArCanReceiver_0.ReceivedFrame.ID = 16#601 THEN

					memcpy(ADR(SubBMS.Rack1.BSA.Rack_Calc.Value), ADR(ArCanReceiver.ArCanReceiver_0.ReceivedFrame.Data), SIZEOF(SubBMS.Rack1.BSA.Rack_Calc.Value));

				END_IF;
				IF ArCanReceiver.ArCanReceiver_0.ReceivedFrame.ID = 16#602 THEN

					memcpy(ADR(SubBMS.Rack1.BSA.Rack_State.Value), ADR(ArCanReceiver.ArCanReceiver_0.ReceivedFrame.Data), SIZEOF(SubBMS.Rack1.BSA.Rack_State.Value));

				END_IF;
				IF ArCanReceiver.ArCanReceiver_0.ReceivedFrame.ID = 16#603 THEN

					memcpy(ADR(SubBMS.Rack1.BSA.Rack_AlarmState.Value), ADR(ArCanReceiver.ArCanReceiver_0.ReceivedFrame.Data), SIZEOF(SubBMS.Rack1.BSA.Rack_AlarmState.Value));

				END_IF;
				IF ArCanReceiver.ArCanReceiver_0.ReceivedFrame.ID = 16#604 THEN

					memcpy(ADR(SubBMS.Rack1.BSA.Rack_PWRCalc.Value), ADR(ArCanReceiver.ArCanReceiver_0.ReceivedFrame.Data), SIZEOF(SubBMS.Rack1.BSA.Rack_PWRCalc.Value));

				END_IF;
				IF ArCanReceiver.ArCanReceiver_0.ReceivedFrame.ID = 16#605 THEN

					memcpy(ADR(SubBMS.Rack1.BSA.Rack_Cell_Vcalc.Value), ADR(ArCanReceiver.ArCanReceiver_0.ReceivedFrame.Data), SIZEOF(SubBMS.Rack1.BSA.Rack_Cell_Vcalc.Value));

				END_IF;
				IF ArCanReceiver.ArCanReceiver_0.ReceivedFrame.ID = 16#606 THEN

					memcpy(ADR(SubBMS.Rack1.BSA.Rack_Cell_Tcalc.Value), ADR(ArCanReceiver.ArCanReceiver_0.ReceivedFrame.Data), SIZEOF(SubBMS.Rack1.BSA.Rack_Cell_Tcalc.Value));

				END_IF;
				IF ArCanReceiver.ArCanReceiver_0.ReceivedFrame.ID = 16#607 THEN

					memcpy(ADR(SubBMS.Rack1.BSA.Rack_Cell_Pcalc.Value), ADR(ArCanReceiver.ArCanReceiver_0.ReceivedFrame.Data), SIZEOF(SubBMS.Rack1.BSA.Rack_Cell_Pcalc.Value));

				END_IF;
				IF ArCanReceiver.ArCanReceiver_0.ReceivedFrame.ID = 16#608 THEN

					memcpy(ADR(SubBMS.Rack1.BSA.Modul1_Info.Value), ADR(ArCanReceiver.ArCanReceiver_0.ReceivedFrame.Data), SIZEOF(SubBMS.Rack1.BSA.Modul1_Info.Value));

				END_IF;
				IF ArCanReceiver.ArCanReceiver_0.ReceivedFrame.ID = 16#609 THEN

					memcpy(ADR(SubBMS.Rack1.BSA.Modul2_Info.Value), ADR(ArCanReceiver.ArCanReceiver_0.ReceivedFrame.Data), SIZEOF(SubBMS.Rack1.BSA.Modul2_Info.Value));

				END_IF;
				IF ArCanReceiver.ArCanReceiver_0.ReceivedFrame.ID = 16#60A THEN

					memcpy(ADR(SubBMS.Rack1.BSA.Modul3_Info.Value), ADR(ArCanReceiver.ArCanReceiver_0.ReceivedFrame.Data), SIZEOF(SubBMS.Rack1.BSA.Modul3_Info.Value));

				END_IF;
				IF ArCanReceiver.ArCanReceiver_0.ReceivedFrame.ID = 16#60B THEN

					memcpy(ADR(SubBMS.Rack1.BSA.Modul4_Info.Value), ADR(ArCanReceiver.ArCanReceiver_0.ReceivedFrame.Data), SIZEOF(SubBMS.Rack1.BSA.Modul4_Info.Value));

				END_IF;
				IF ArCanReceiver.ArCanReceiver_0.ReceivedFrame.ID = 16#60C THEN

					memcpy(ADR(SubBMS.Rack1.BSA.Modul5_Info.Value), ADR(ArCanReceiver.ArCanReceiver_0.ReceivedFrame.Data), SIZEOF(SubBMS.Rack1.BSA.Modul5_Info.Value));

				END_IF;
				IF ArCanReceiver.ArCanReceiver_0.ReceivedFrame.ID = 16#60D THEN

					memcpy(ADR(SubBMS.Rack1.BSA.Modul6_Info.Value), ADR(ArCanReceiver.ArCanReceiver_0.ReceivedFrame.Data), SIZEOF(SubBMS.Rack1.BSA.Modul6_Info.Value));

				END_IF;
				IF ArCanReceiver.ArCanReceiver_0.ReceivedFrame.ID = 16#60E THEN

					memcpy(ADR(SubBMS.Rack1.BSA.Modul7_Info.Value), ADR(ArCanReceiver.ArCanReceiver_0.ReceivedFrame.Data), SIZEOF(SubBMS.Rack1.BSA.Modul7_Info.Value));

				END_IF;

				16#610..16#61E: // RACK 2

				IF ArCanReceiver.ArCanReceiver_0.ReceivedFrame.ID = 16#610 THEN

					memcpy(ADR(SubBMS.Rack2.BSA.BSA_Product.Value), ADR(ArCanReceiver.ArCanReceiver_0.ReceivedFrame.Data), SIZEOF(SubBMS.Rack2.BSA.BSA_Product.Value));

				END_IF;
				IF ArCanReceiver.ArCanReceiver_0.ReceivedFrame.ID = 16#611 THEN

					memcpy(ADR(SubBMS.Rack2.BSA.Rack_Calc.Value), ADR(ArCanReceiver.ArCanReceiver_0.ReceivedFrame.Data), SIZEOF(SubBMS.Rack2.BSA.Rack_Calc.Value));

				END_IF;
				IF ArCanReceiver.ArCanReceiver_0.ReceivedFrame.ID = 16#612 THEN

					memcpy(ADR(SubBMS.Rack2.BSA.Rack_State.Value), ADR(ArCanReceiver.ArCanReceiver_0.ReceivedFrame.Data), SIZEOF(SubBMS.Rack2.BSA.Rack_State.Value));

				END_IF;
				IF ArCanReceiver.ArCanReceiver_0.ReceivedFrame.ID = 16#613 THEN

					memcpy(ADR(SubBMS.Rack2.BSA.Rack_AlarmState.Value), ADR(ArCanReceiver.ArCanReceiver_0.ReceivedFrame.Data), SIZEOF(SubBMS.Rack2.BSA.Rack_AlarmState.Value));

				END_IF;
				IF ArCanReceiver.ArCanReceiver_0.ReceivedFrame.ID = 16#614 THEN

					memcpy(ADR(SubBMS.Rack2.BSA.Rack_PWRCalc.Value), ADR(ArCanReceiver.ArCanReceiver_0.ReceivedFrame.Data), SIZEOF(SubBMS.Rack2.BSA.Rack_PWRCalc.Value));

				END_IF;
				IF ArCanReceiver.ArCanReceiver_0.ReceivedFrame.ID = 16#615 THEN

					memcpy(ADR(SubBMS.Rack2.BSA.Rack_Cell_Vcalc.Value), ADR(ArCanReceiver.ArCanReceiver_0.ReceivedFrame.Data), SIZEOF(SubBMS.Rack2.BSA.Rack_Cell_Vcalc.Value));

				END_IF;
				IF ArCanReceiver.ArCanReceiver_0.ReceivedFrame.ID = 16#616 THEN

					memcpy(ADR(SubBMS.Rack2.BSA.Rack_Cell_Tcalc.Value), ADR(ArCanReceiver.ArCanReceiver_0.ReceivedFrame.Data), SIZEOF(SubBMS.Rack2.BSA.Rack_Cell_Tcalc.Value));

				END_IF;
				IF ArCanReceiver.ArCanReceiver_0.ReceivedFrame.ID = 16#617 THEN

					memcpy(ADR(SubBMS.Rack2.BSA.Rack_Cell_Pcalc.Value), ADR(ArCanReceiver.ArCanReceiver_0.ReceivedFrame.Data), SIZEOF(SubBMS.Rack2.BSA.Rack_Cell_Pcalc.Value));

				END_IF;
				IF ArCanReceiver.ArCanReceiver_0.ReceivedFrame.ID = 16#618 THEN

					memcpy(ADR(SubBMS.Rack2.BSA.Modul1_Info.Value), ADR(ArCanReceiver.ArCanReceiver_0.ReceivedFrame.Data), SIZEOF(SubBMS.Rack2.BSA.Modul1_Info.Value));

				END_IF;
				IF ArCanReceiver.ArCanReceiver_0.ReceivedFrame.ID = 16#619 THEN

					memcpy(ADR(SubBMS.Rack2.BSA.Modul2_Info.Value), ADR(ArCanReceiver.ArCanReceiver_0.ReceivedFrame.Data), SIZEOF(SubBMS.Rack2.BSA.Modul2_Info.Value));

				END_IF;
				IF ArCanReceiver.ArCanReceiver_0.ReceivedFrame.ID = 16#61A THEN

					memcpy(ADR(SubBMS.Rack2.BSA.Modul3_Info.Value), ADR(ArCanReceiver.ArCanReceiver_0.ReceivedFrame.Data), SIZEOF(SubBMS.Rack2.BSA.Modul3_Info.Value));

				END_IF;
				IF ArCanReceiver.ArCanReceiver_0.ReceivedFrame.ID = 16#61B THEN

					memcpy(ADR(SubBMS.Rack2.BSA.Modul4_Info.Value), ADR(ArCanReceiver.ArCanReceiver_0.ReceivedFrame.Data), SIZEOF(SubBMS.Rack2.BSA.Modul4_Info.Value));

				END_IF;
				IF ArCanReceiver.ArCanReceiver_0.ReceivedFrame.ID = 16#61C THEN

					memcpy(ADR(SubBMS.Rack2.BSA.Modul5_Info.Value), ADR(ArCanReceiver.ArCanReceiver_0.ReceivedFrame.Data), SIZEOF(SubBMS.Rack2.BSA.Modul5_Info.Value));

				END_IF;
				IF ArCanReceiver.ArCanReceiver_0.ReceivedFrame.ID = 16#61D THEN

					memcpy(ADR(SubBMS.Rack2.BSA.Modul6_Info.Value), ADR(ArCanReceiver.ArCanReceiver_0.ReceivedFrame.Data), SIZEOF(SubBMS.Rack2.BSA.Modul6_Info.Value));

				END_IF;
				IF ArCanReceiver.ArCanReceiver_0.ReceivedFrame.ID = 16#61E THEN

					memcpy(ADR(SubBMS.Rack2.BSA.Modul7_Info.Value), ADR(ArCanReceiver.ArCanReceiver_0.ReceivedFrame.Data), SIZEOF(SubBMS.Rack2.BSA.Modul7_Info.Value));

				END_IF;

				16#620..16#62E: // RACK 2

				IF ArCanReceiver.ArCanReceiver_0.ReceivedFrame.ID = 16#620 THEN

					memcpy(ADR(SubBMS.Rack3.BSA.BSA_Product.Value), ADR(ArCanReceiver.ArCanReceiver_0.ReceivedFrame.Data), SIZEOF(SubBMS.Rack3.BSA.BSA_Product.Value));

				END_IF;
				IF ArCanReceiver.ArCanReceiver_0.ReceivedFrame.ID = 16#621 THEN

					memcpy(ADR(SubBMS.Rack3.BSA.Rack_Calc.Value), ADR(ArCanReceiver.ArCanReceiver_0.ReceivedFrame.Data), SIZEOF(SubBMS.Rack3.BSA.Rack_Calc.Value));

				END_IF;
				IF ArCanReceiver.ArCanReceiver_0.ReceivedFrame.ID = 16#622 THEN

					memcpy(ADR(SubBMS.Rack3.BSA.Rack_State.Value), ADR(ArCanReceiver.ArCanReceiver_0.ReceivedFrame.Data), SIZEOF(SubBMS.Rack3.BSA.Rack_State.Value));

				END_IF;
				IF ArCanReceiver.ArCanReceiver_0.ReceivedFrame.ID = 16#623 THEN

					memcpy(ADR(SubBMS.Rack3.BSA.Rack_AlarmState.Value), ADR(ArCanReceiver.ArCanReceiver_0.ReceivedFrame.Data), SIZEOF(SubBMS.Rack3.BSA.Rack_AlarmState.Value));

				END_IF;
				IF ArCanReceiver.ArCanReceiver_0.ReceivedFrame.ID = 16#624 THEN

					memcpy(ADR(SubBMS.Rack3.BSA.Rack_PWRCalc.Value), ADR(ArCanReceiver.ArCanReceiver_0.ReceivedFrame.Data), SIZEOF(SubBMS.Rack3.BSA.Rack_PWRCalc.Value));

				END_IF;
				IF ArCanReceiver.ArCanReceiver_0.ReceivedFrame.ID = 16#625 THEN

					memcpy(ADR(SubBMS.Rack3.BSA.Rack_Cell_Vcalc.Value), ADR(ArCanReceiver.ArCanReceiver_0.ReceivedFrame.Data), SIZEOF(SubBMS.Rack3.BSA.Rack_Cell_Vcalc.Value));

				END_IF;
				IF ArCanReceiver.ArCanReceiver_0.ReceivedFrame.ID = 16#626 THEN

					memcpy(ADR(SubBMS.Rack3.BSA.Rack_Cell_Tcalc.Value), ADR(ArCanReceiver.ArCanReceiver_0.ReceivedFrame.Data), SIZEOF(SubBMS.Rack3.BSA.Rack_Cell_Tcalc.Value));

				END_IF;
				IF ArCanReceiver.ArCanReceiver_0.ReceivedFrame.ID = 16#627 THEN

					memcpy(ADR(SubBMS.Rack3.BSA.Rack_Cell_Pcalc.Value), ADR(ArCanReceiver.ArCanReceiver_0.ReceivedFrame.Data), SIZEOF(SubBMS.Rack3.BSA.Rack_Cell_Pcalc.Value));

				END_IF;
				IF ArCanReceiver.ArCanReceiver_0.ReceivedFrame.ID = 16#628 THEN

					memcpy(ADR(SubBMS.Rack3.BSA.Modul1_Info.Value), ADR(ArCanReceiver.ArCanReceiver_0.ReceivedFrame.Data), SIZEOF(SubBMS.Rack3.BSA.Modul1_Info.Value));

				END_IF;
				IF ArCanReceiver.ArCanReceiver_0.ReceivedFrame.ID = 16#629 THEN

					memcpy(ADR(SubBMS.Rack3.BSA.Modul2_Info.Value), ADR(ArCanReceiver.ArCanReceiver_0.ReceivedFrame.Data), SIZEOF(SubBMS.Rack3.BSA.Modul2_Info.Value));

				END_IF;
				IF ArCanReceiver.ArCanReceiver_0.ReceivedFrame.ID = 16#62A THEN

					memcpy(ADR(SubBMS.Rack3.BSA.Modul3_Info.Value), ADR(ArCanReceiver.ArCanReceiver_0.ReceivedFrame.Data), SIZEOF(SubBMS.Rack3.BSA.Modul3_Info.Value));

				END_IF;
				IF ArCanReceiver.ArCanReceiver_0.ReceivedFrame.ID = 16#62B THEN

					memcpy(ADR(SubBMS.Rack3.BSA.Modul4_Info.Value), ADR(ArCanReceiver.ArCanReceiver_0.ReceivedFrame.Data), SIZEOF(SubBMS.Rack3.BSA.Modul4_Info.Value));

				END_IF;
				IF ArCanReceiver.ArCanReceiver_0.ReceivedFrame.ID = 16#62C THEN

					memcpy(ADR(SubBMS.Rack3.BSA.Modul5_Info.Value), ADR(ArCanReceiver.ArCanReceiver_0.ReceivedFrame.Data), SIZEOF(SubBMS.Rack3.BSA.Modul5_Info.Value));

				END_IF;
				IF ArCanReceiver.ArCanReceiver_0.ReceivedFrame.ID = 16#62D THEN

					memcpy(ADR(SubBMS.Rack3.BSA.Modul6_Info.Value), ADR(ArCanReceiver.ArCanReceiver_0.ReceivedFrame.Data), SIZEOF(SubBMS.Rack3.BSA.Modul6_Info.Value));

				END_IF;
				IF ArCanReceiver.ArCanReceiver_0.ReceivedFrame.ID = 16#62E THEN

					memcpy(ADR(SubBMS.Rack3.BSA.Modul7_Info.Value), ADR(ArCanReceiver.ArCanReceiver_0.ReceivedFrame.Data), SIZEOF(SubBMS.Rack3.BSA.Modul7_Info.Value));

				END_IF;
				16#630..16#63E: // RACK 2

				IF ArCanReceiver.ArCanReceiver_0.ReceivedFrame.ID = 16#630 THEN

					memcpy(ADR(SubBMS.Rack4.BSA.BSA_Product.Value), ADR(ArCanReceiver.ArCanReceiver_0.ReceivedFrame.Data), SIZEOF(SubBMS.Rack4.BSA.BSA_Product.Value));

				END_IF;
				IF ArCanReceiver.ArCanReceiver_0.ReceivedFrame.ID = 16#631 THEN

					memcpy(ADR(SubBMS.Rack4.BSA.Rack_Calc.Value), ADR(ArCanReceiver.ArCanReceiver_0.ReceivedFrame.Data), SIZEOF(SubBMS.Rack4.BSA.Rack_Calc.Value));

				END_IF;
				IF ArCanReceiver.ArCanReceiver_0.ReceivedFrame.ID = 16#632 THEN

					memcpy(ADR(SubBMS.Rack4.BSA.Rack_State.Value), ADR(ArCanReceiver.ArCanReceiver_0.ReceivedFrame.Data), SIZEOF(SubBMS.Rack4.BSA.Rack_State.Value));

				END_IF;
				IF ArCanReceiver.ArCanReceiver_0.ReceivedFrame.ID = 16#633 THEN

					memcpy(ADR(SubBMS.Rack4.BSA.Rack_AlarmState.Value), ADR(ArCanReceiver.ArCanReceiver_0.ReceivedFrame.Data), SIZEOF(SubBMS.Rack4.BSA.Rack_AlarmState.Value));

				END_IF;
				IF ArCanReceiver.ArCanReceiver_0.ReceivedFrame.ID = 16#634 THEN

					memcpy(ADR(SubBMS.Rack4.BSA.Rack_PWRCalc.Value), ADR(ArCanReceiver.ArCanReceiver_0.ReceivedFrame.Data), SIZEOF(SubBMS.Rack4.BSA.Rack_PWRCalc.Value));

				END_IF;
				IF ArCanReceiver.ArCanReceiver_0.ReceivedFrame.ID = 16#635 THEN

					memcpy(ADR(SubBMS.Rack4.BSA.Rack_Cell_Vcalc.Value), ADR(ArCanReceiver.ArCanReceiver_0.ReceivedFrame.Data), SIZEOF(SubBMS.Rack4.BSA.Rack_Cell_Vcalc.Value));

				END_IF;
				IF ArCanReceiver.ArCanReceiver_0.ReceivedFrame.ID = 16#636 THEN

					memcpy(ADR(SubBMS.Rack4.BSA.Rack_Cell_Tcalc.Value), ADR(ArCanReceiver.ArCanReceiver_0.ReceivedFrame.Data), SIZEOF(SubBMS.Rack4.BSA.Rack_Cell_Tcalc.Value));

				END_IF;
				IF ArCanReceiver.ArCanReceiver_0.ReceivedFrame.ID = 16#637 THEN

					memcpy(ADR(SubBMS.Rack4.BSA.Rack_Cell_Pcalc.Value), ADR(ArCanReceiver.ArCanReceiver_0.ReceivedFrame.Data), SIZEOF(SubBMS.Rack4.BSA.Rack_Cell_Pcalc.Value));

				END_IF;
				IF ArCanReceiver.ArCanReceiver_0.ReceivedFrame.ID = 16#638 THEN

					memcpy(ADR(SubBMS.Rack4.BSA.Modul1_Info.Value), ADR(ArCanReceiver.ArCanReceiver_0.ReceivedFrame.Data), SIZEOF(SubBMS.Rack4.BSA.Modul1_Info.Value));

				END_IF;
				IF ArCanReceiver.ArCanReceiver_0.ReceivedFrame.ID = 16#639 THEN

					memcpy(ADR(SubBMS.Rack4.BSA.Modul2_Info.Value), ADR(ArCanReceiver.ArCanReceiver_0.ReceivedFrame.Data), SIZEOF(SubBMS.Rack4.BSA.Modul2_Info.Value));

				END_IF;
				IF ArCanReceiver.ArCanReceiver_0.ReceivedFrame.ID = 16#63A THEN

					memcpy(ADR(SubBMS.Rack4.BSA.Modul3_Info.Value), ADR(ArCanReceiver.ArCanReceiver_0.ReceivedFrame.Data), SIZEOF(SubBMS.Rack4.BSA.Modul3_Info.Value));

				END_IF;
				IF ArCanReceiver.ArCanReceiver_0.ReceivedFrame.ID = 16#63B THEN

					memcpy(ADR(SubBMS.Rack4.BSA.Modul4_Info.Value), ADR(ArCanReceiver.ArCanReceiver_0.ReceivedFrame.Data), SIZEOF(SubBMS.Rack4.BSA.Modul4_Info.Value));

				END_IF;
				IF ArCanReceiver.ArCanReceiver_0.ReceivedFrame.ID = 16#63C THEN

					memcpy(ADR(SubBMS.Rack4.BSA.Modul5_Info.Value), ADR(ArCanReceiver.ArCanReceiver_0.ReceivedFrame.Data), SIZEOF(SubBMS.Rack4.BSA.Modul5_Info.Value));

				END_IF;
				IF ArCanReceiver.ArCanReceiver_0.ReceivedFrame.ID = 16#63D THEN

					memcpy(ADR(SubBMS.Rack4.BSA.Modul6_Info.Value), ADR(ArCanReceiver.ArCanReceiver_0.ReceivedFrame.Data), SIZEOF(SubBMS.Rack4.BSA.Modul6_Info.Value));

				END_IF;
				IF ArCanReceiver.ArCanReceiver_0.ReceivedFrame.ID = 16#63E THEN

					memcpy(ADR(SubBMS.Rack4.BSA.Modul7_Info.Value), ADR(ArCanReceiver.ArCanReceiver_0.ReceivedFrame.Data), SIZEOF(SubBMS.Rack4.BSA.Modul7_Info.Value));

				END_IF;

			END_CASE;

		END_IF

		ActRACK1DATARxParshing;
		ActRACK2DATARxParshing;
		ActRACK3DATARxParshing;
		ActRACK4DATARxParshing;

		(***********************************************************)
		(* CAN Communication Status *)
		(***********************************************************)

		IF ArCanReceiver.ArCanReceiver_0.Error THEN
			gComm.CAN1.bError	:= TRUE;
			gComm.CAN1.bActive	:= FALSE;
			gComm.CAN1.bTransmitting	:= FALSE;
		ELSIF ArCanReceiver.ArCanReceiver_0.Active AND ArCanReceiver.ArCanReceiver_0.Busy THEN
			gComm.CAN1.bError	:= FALSE;
			gComm.CAN1.bActive	:= TRUE;

			IF (countCANSuccessOld <> ArCanReceiver.successCount) THEN
				countCANSuccessOld	:= ArCanReceiver.successCount;
				gComm.CAN1.bTransmitting	:= TRUE;
				countTime	:= 0;
			ELSE
				countTime	:= countTime + 1;
				IF (countTime > 50) THEN
					gComm.CAN1.bTransmitting	:= FALSE;
					countTime	:= 0;
				END_IF
			END_IF
		ELSE
			gComm.CAN1.bError	:= FALSE;
			gComm.CAN1.bActive	:= FALSE;
			gComm.CAN1.bTransmitting	:= FALSE;
		END_IF
		(***********************************************************)
	END_IF;

END_PROGRAM

PROGRAM _EXIT

(* Deinitialization of the receiver *)
	ArCanReceiver.ArCanReceiver_0.Enable	:= FALSE;
	ArCanReceiver.ArCanReceiver_0();

END_PROGRAM
```

#### ArCanReceive.var - Local variables
```iecst
VAR
	ArCanReceiver : ArCanReceive_typ;
	countTime : USINT;
	countCANSuccessOld : UDINT;
	CmdSim : BOOL;
END_VAR
```

#### CanReceiver.st
```iecst
ACTION ActArCanReceiver:

	CASE ArCanReceiver.step OF
		STEP_WAIT:
			(* wait for starting *)
			IF ArCanReceiver.enable = TRUE THEN
				ArCanReceiver.step	:= STEP_INIT_BAUDRATE;
			END_IF

		STEP_INIT_BAUDRATE:	(* Initializes the receiver with ArCanSetBitTimingRegisters to 250 kbit/s *)
			ArCanReceiver.ArCanSetBitTimingRegisters_0.Execute := TRUE;
			ArCanReceiver.ArCanSetBitTimingRegisters_0.DeviceName := ArCanReceiver.receiverDeviceName;
			//			ArCanReceiver.ArCanSetBitTimingRegisters_0.Register0 := 1;	(* Set to 250 000 bit/s *)
			//			ArCanReceiver.ArCanSetBitTimingRegisters_0.Register1 := 28;	(* Set to 250 000 bit/s *)

			ArCanReceiver.ArCanSetBitTimingRegisters_0();

			IF (ArCanReceiver.ArCanSetBitTimingRegisters_0.Done = TRUE) THEN
				gSignalCheck.Can_HardwareCheck2 := TRUE;
				ArCanReceiver.step := STEP_INIT_RECEIVER;
			ELSIF (ArCanReceiver.ArCanSetBitTimingRegisters_0.Error = TRUE) THEN
				ArCanReceiver.lastError := ArCanReceiver.ArCanSetBitTimingRegisters_0.StatusID;
				ArCanReceiver.errorCount := ArCanReceiver.errorCount + 1;
				ArCanReceiver.step := STEP_ERROR;
			END_IF;

		STEP_INIT_RECEIVER:	(* Initializes the CAN Receiver *)
			ArCanReceiver.ArCanReceiver_0.Enable := TRUE;			(* FALSE -> TRUE takeovers the input parameters *)
			ArCanReceiver.ArCanReceiver_0.DeviceName := ArCanReceiver.receiverDeviceName;
			ArCanReceiver.ArCanReceiver_0.ID := ArCanReceiver.id;				(* dummy, because IDMask is arCAN_RECEIVE_ALL *)
			ArCanReceiver.ArCanReceiver_0.IDMask := ArCanReceiver.idMask;
			ArCanReceiver.ArCanReceiver_0.Format := ArCanReceiver.format;
			ArCanReceiver.ArCanReceiver_0.QueueSize	:= ArCanReceiver.queueSize;

			IF (ArCanReceiver.ArCanReceiver_0.Active = TRUE) THEN

				gSignalCheck.Can_ReceiveCheck := TRUE;
				ArCanReceiver.step := STEP_WAIT_FOR_DATA;
			ELSIF (ArCanReceiver.ArCanReceiver_0.Error = TRUE) THEN
				ArCanReceiver.errorCount := ArCanReceiver.errorCount + 1;
				ArCanReceiver.lastError := ArCanReceiver.ArCanReceiver_0.StatusID;
				ArCanReceiver.step := STEP_ERROR;
			END_IF;

		STEP_WAIT_FOR_DATA:	(* Checks for new data *)
			IF (ArCanReceiver.ArCanReceiver_0.NewDataValid) THEN
				ArCanReceiver.successCount := ArCanReceiver.successCount + 1;

				(* copy received data & save timestamp *)
				memcpy( ADR(ArCanReceiver.receivedIterationCounter), ADR(ArCanReceiver.ArCanReceiver_0.ReceivedFrame), SIZEOF(ArCanReceiver.receivedIterationCounter));

				ArCanReceiver.lastReceiveTimestamp := ArCanReceiver.ArCanReceiver_0.Timestamp.UTCSeconds;

				ArCanReceiver.lostFrames := ArCanReceiver.lostFrames + ArCanReceiver.ArCanReceiver_0.NumberOfLostFrames;
			ELSIF (ArCanReceiver.ArCanReceiver_0.Error) THEN
				ArCanReceiver.errorCount := ArCanReceiver.errorCount + 1;
				ArCanReceiver.lastError := ArCanReceiver.ArCanReceiver_0.StatusID;
				ArCanReceiver.step := STEP_ERROR;
			ELSE
				memset( ADR(ArCanReceiver.ArCanReceiver_0.ReceivedFrame.ID), 0, SIZEOF(ArCanReceiver.ArCanReceiver_0.ReceivedFrame.ID));
			END_IF;

			IF (ArCanReceiver.enable = FALSE) THEN (* User stops the test *)
				ArCanReceiver.step := STEP_DEINIT;
			END_IF;

		STEP_DEINIT:
			ArCanReceiver.ArCanReceiver_0.Enable := FALSE;
			ArCanReceiver.step := STEP_WAIT;

		STEP_ERROR:
			ArCanReceiver.ArCanReceiver_0.Enable := FALSE;
			ArCanReceiver.step := STEP_WAIT;
		ELSE

	END_CASE;

	ArCanReceiver.ArCanReceiver_0();

END_ACTION
```
